LIN {X 0,Y 531.012,Z 558.342,A -85,B 0,C 180,E1 -4347.596,E2 -4347.596} C_VEL
LIN {X 0,Y 530.977,Z 558.347,A -85,B 0,C 180,E1 -4350.648,E2 -4350.648} C_VEL
LIN {X 0,Y 530.988,Z 558.345,A -85,B 0,C 180,E1 -4353.773,E2 -4353.773} C_VEL
LIN {X 0,Y 530.967,Z 558.348,A -85,B 0,C 180,E1 -4356.558,E2 -4356.558} C_VEL
LIN {X 0,Y 531.002,Z 558.343,A -85,B 0,C 180,E1 -4359.858,E2 -4359.858} C_VEL
LIN {X 0,Y 530.979,Z 558.345,A -85,B 0,C 180,E1 -4362.457,E2 -4362.457} C_VEL
LIN {X 0,Y 530.984,Z 558.347,A -85,B 0,C 180,E1 -4365.622,E2 -4365.622} C_VEL
LIN {X 0,Y 531.004,Z 558.343,A -85,B 0,C 180,E1 -4368.567,E2 -4368.567} C_VEL
LIN {X 0,Y 530.967,Z 558.349,A -85,B 0,C 180,E1 -4371.347,E2 -4371.347} C_VEL
LIN {X 0,Y 530.976,Z 558.441,A -85,B 0,C 180,E1 -4371.895,E2 -4371.895} C_VEL
LIN {X 0,Y 532.393,Z 565.517,A -85,B 0,C 180,E1 -4373.635,E2 -4373.635} C_VEL
LIN {X 0,Y 532.607,Z 569.285,A -85,B 0,C 180,E1 -4374.508,E2 -4374.508} C_VEL
LIN {X 0,Y 532.356,Z 582.925,A -85,B 0,C 180,E1 -4377.495,E2 -4377.495} C_VEL
LIN {X 0,Y 532.166,Z 596.383,A -85,B 0,C 180,E1 -4380.31,E2 -4380.31} C_VEL
LIN {X 0,Y 531.962,Z 611.243,A -85,B 0,C 180,E1 -4383.309,E2 -4383.309} C_VEL
LIN {X 0,Y 531.773,Z 627.111,A -85,B 0,C 180,E1 -4386.436,E2 -4386.436} C_VEL
LIN {X 0,Y 531.567,Z 641.948,A -85,B 0,C 180,E1 -4389.289,E2 -4389.289} C_VEL
LIN {X 0,Y 531.378,Z 654.54,A -85,B 0,C 180,E1 -4391.713,E2 -4391.713} C_VEL
LIN {X 0,Y 531.087,Z 669.174,A -85,B 0,C 180,E1 -4394.654,E2 -4394.654} C_VEL
LIN {X 0,Y 530.95,Z 678.137,A -85,B 0,C 180,E1 -4396.436,E2 -4396.436} C_VEL
LIN {X 0,Y 532.382,Z 688.546,A -85,B 0,C 180,E1 -4396.668,E2 -4396.668} C_VEL
LIN {X 0,Y 532.174,Z 700.896,A -85,B 0,C 180,E1 -4397.027,E2 -4397.027} C_VEL
LIN {X 0,Y 531.979,Z 712.521,A -85,B 0,C 180,E1 -4397.507,E2 -4397.507} C_VEL
LIN {X 0,Y 531.678,Z 724.909,A -85,B 0,C 180,E1 -4398.185,E2 -4398.185} C_VEL
LIN {X 0,Y 531.5,Z 735.754,A -85,B 0,C 180,E1 -4398.947,E2 -4398.947} C_VEL
LIN {X 0,Y 531.189,Z 746.607,A -85,B 0,C 180,E1 -4399.904,E2 -4399.904} C_VEL
LIN {X 0,Y 530.969,Z 755.419,A -85,B 0,C 180,E1 -4400.862,E2 -4400.862} C_VEL
LIN {X 0,Y 530.779,Z 764.008,A -85,B 0,C 180,E1 -4402.009,E2 -4402.009} C_VEL
LIN {X 0,Y 530.636,Z 770.872,A -85,B 0,C 180,E1 -4403.155,E2 -4403.155} C_VEL
LIN {X 0,Y 530.611,Z 776.369,A -85,B 0,C 180,E1 -4404.3,E2 -4404.3} C_VEL
LIN {X 0,Y 530.457,Z 780.679,A -85,B 0,C 180,E1 -4405.441,E2 -4405.441} C_VEL
LIN {X 0,Y 530.516,Z 782.96,A -85,B 0,C 180,E1 -4406.203,E2 -4406.203} C_VEL
LIN {X 0,Y 530.457,Z 784.809,A -85,B 0,C 180,E1 -4406.963,E2 -4406.963} C_VEL
LIN {X 0,Y 530.41,Z 786.196,A -85,B 0,C 180,E1 -4407.723,E2 -4407.723} C_VEL
LIN {X 0,Y 530.344,Z 787.786,A -85,B 0,C 180,E1 -4409.241,E2 -4409.241} C_VEL
LIN {X 0,Y 530.342,Z 788,A -85,B 0,C 180,E1 -4410.001,E2 -4410.001} C_VEL
LIN {X 0,Y 530.361,Z 787.184,A -85,B 0,C 180,E1 -4411.519,E2 -4411.519} C_VEL
LIN {X 0,Y 530.41,Z 786.196,A -85,B 0,C 180,E1 -4412.279,E2 -4412.279} C_VEL
LIN {X 0,Y 530.457,Z 784.809,A -85,B 0,C 180,E1 -4413.039,E2 -4413.039} C_VEL
LIN {X 0,Y 530.523,Z 781.893,A -85,B 0,C 180,E1 -4414.179,E2 -4414.179} C_VEL
LIN {X 0,Y 530.525,Z 777.946,A -85,B 0,C 180,E1 -4415.321,E2 -4415.321} C_VEL
LIN {X 0,Y 530.6,Z 772.262,A -85,B 0,C 180,E1 -4416.582,E2 -4416.582} C_VEL
LIN {X 0,Y 530.759,Z 765.232,A -85,B 0,C 180,E1 -4417.801,E2 -4417.801} C_VEL
LIN {X 0,Y 530.93,Z 756.987,A -85,B 0,C 180,E1 -4418.949,E2 -4418.949} C_VEL
LIN {X 0,Y 531.112,Z 748.533,A -85,B 0,C 180,E1 -4419.906,E2 -4419.906} C_VEL
LIN {X 0,Y 531.416,Z 738.086,A -85,B 0,C 180,E1 -4420.863,E2 -4420.863} C_VEL
LIN {X 0,Y 531.675,Z 727.295,A -85,B 0,C 180,E1 -4421.66,E2 -4421.66} C_VEL
LIN {X 0,Y 531.876,Z 716.394,A -85,B 0,C 180,E1 -4422.303,E2 -4422.303} C_VEL
LIN {X 0,Y 532.111,Z 704.747,A -85,B 0,C 180,E1 -4422.83,E2 -4422.83} C_VEL
LIN {X 0,Y 532.332,Z 691.322,A -85,B 0,C 180,E1 -4423.262,E2 -4423.262} C_VEL
LIN {X 0,Y 532.131,Z 685.757,A -85,B 0,C 180,E1 -4423.398,E2 -4423.398} C_VEL
LIN {X 0,Y 530.944,Z 678.031,A -85,B 0,C 180,E1 -4423.589,E2 -4423.589} C_VEL
LIN {X 0,Y 531.198,Z 663.358,A -85,B 0,C 180,E1 -4426.527,E2 -4426.527} C_VEL
LIN {X 0,Y 531.508,Z 648.458,A -85,B 0,C 180,E1 -4429.505,E2 -4429.505} C_VEL
LIN {X 0,Y 531.685,Z 632.611,A -85,B 0,C 180,E1 -4432.541,E2 -4432.541} C_VEL
LIN {X 0,Y 531.884,Z 617.998,A -85,B 0,C 180,E1 -4435.432,E2 -4435.432} C_VEL
LIN {X 0,Y 532.057,Z 605.161,A -85,B 0,C 180,E1 -4438.028,E2 -4438.028} C_VEL
LIN {X 0,Y 532.312,Z 590.837,A -85,B 0,C 180,E1 -4440.992,E2 -4440.992} C_VEL
LIN {X 0,Y 532.502,Z 577.979,A -85,B 0,C 180,E1 -4443.749,E2 -4443.749} C_VEL
LIN {X 0,Y 532.673,Z 568.114,A -85,B 0,C 180,E1 -4445.926,E2 -4445.926} C_VEL
LIN {X 0,Y 531.615,Z 561.406,A -85,B 0,C 180,E1 -4447.514,E2 -4447.514} C_VEL
LIN {X 0,Y 530.971,Z 558.349,A -85,B 0,C 180,E1 -4448.288,E2 -4448.288} C_VEL
LIN {X 0,Y 531.006,Z 558.343,A -85,B 0,C 180,E1 -4451.435,E2 -4451.435} C_VEL
LIN {X 0,Y 530.993,Z 558.346,A -85,B 0,C 180,E1 -4454.547,E2 -4454.547} C_VEL
LIN {X 0,Y 530.99,Z 558.346,A -85,B 0,C 180,E1 -4457.834,E2 -4457.834} C_VEL
LIN {X 0,Y 530.99,Z 558.344,A -85,B 0,C 180,E1 -4460.557,E2 -4460.557} C_VEL
LIN {X 0,Y 530.979,Z 558.347,A -85,B 0,C 180,E1 -4463.842,E2 -4463.842} C_VEL
LIN {X 0,Y 531.004,Z 558.342,A -85,B 0,C 180,E1 -4466.494,E2 -4466.494} C_VEL
LIN {X 0,Y 530.978,Z 558.346,A -85,B 0,C 180,E1 -4469.355,E2 -4469.355} C_VEL
LIN {X 0,Y 531.021,Z 558.34,A -85,B 0,C 180,E1 -4472.467,E2 -4472.467} C_VEL
LIN {X 0,Y 531.01,Z 558.341,A -85,B 0,C 180,E1 -4474.942,E2 -4474.942} C_VEL
LIN {X 0,Y 530.976,Z 558.346,A -85,B 0,C 180,E1 -4478.247,E2 -4478.247} C_VEL
LIN {X 0,Y 530.999,Z 558.343,A -85,B 0,C 180,E1 -4480.677,E2 -4480.677} C_VEL
LIN {X 0,Y 530.99,Z 558.343,A -85,B 0,C 180,E1 -4483.071,E2 -4483.071} C_VEL
LIN {X 0,Y 531.023,Z 558.338,A -85,B 0,C 180,E1 -4485.436,E2 -4485.436} C_VEL
LIN {X 0,Y 531.04,Z 558.339,A -85,B 0,C 180,E1 -4488.55,E2 -4488.55} C_VEL
LIN {X 0,Y 531.061,Z 558.335,A -85,B 0,C 180,E1 -4491.629,E2 -4491.629} C_VEL
LIN {X 0,Y 531.126,Z 558.327,A -85,B 0,C 180,E1 -4494.685,E2 -4494.685} C_VEL
LIN {X 0,Y 531.139,Z 558.327,A -85,B 0,C 180,E1 -4497.725,E2 -4497.725} C_VEL
LIN {X 0,Y 531.157,Z 558.324,A -85,B 0,C 180,E1 -4500.758,E2 -4500.758} C_VEL
LIN {X 0,Y 531.107,Z 558.329,A -85,B 0,C 180,E1 -4503.034,E2 -4503.034} C_VEL
LIN {X 0,Y 531.088,Z 558.333,A -85,B 0,C 180,E1 -4506.077,E2 -4506.077} C_VEL
LIN {X 0,Y 531.031,Z 558.34,A -85,B 0,C 180,E1 -4509.138,E2 -4509.138} C_VEL
LIN {X 0,Y 531.044,Z 558.337,A -85,B 0,C 180,E1 -4512.225,E2 -4512.225} C_VEL
LIN {X 0,Y 530.999,Z 558.343,A -85,B 0,C 180,E1 -4515.349,E2 -4515.349} C_VEL
LIN {X 0,Y 530.993,Z 558.345,A -85,B 0,C 180,E1 -4518.521,E2 -4518.521} C_VEL
LIN {X 0,Y 531.002,Z 558.345,A -85,B 0,C 180,E1 -4520.937,E2 -4520.937} C_VEL
LIN {X 0,Y 530.983,Z 558.345,A -85,B 0,C 180,E1 -4524.224,E2 -4524.224} C_VEL
LIN {X 0,Y 531.008,Z 558.344,A -85,B 0,C 180,E1 -4526.743,E2 -4526.743} C_VEL
LIN {X 0,Y 530.984,Z 558.345,A -85,B 0,C 180,E1 -4529.322,E2 -4529.322} C_VEL
LIN {X 0,Y 530.972,Z 558.346,A -85,B 0,C 180,E1 -4532.101,E2 -4532.101} C_VEL
LIN {X 0,Y 530.99,Z 558.346,A -85,B 0,C 180,E1 -4534.854,E2 -4534.854} C_VEL
LIN {X 0,Y 530.968,Z 558.348,A -85,B 0,C 180,E1 -4537.507,E2 -4537.507} C_VEL
LIN {X 0,Y 530.985,Z 558.345,A -85,B 0,C 180,E1 -4540.432,E2 -4540.432} C_VEL
LIN {X 0,Y 530.972,Z 558.347,A -85,B 0,C 180,E1 -4543.282,E2 -4543.282} C_VEL
LIN {X 0,Y 530.965,Z 558.347,A -85,B 0,C 180,E1 -4543.565,E2 -4543.565} C_VEL
LIN {X 0,Y 530.292,Z 558.433,A -85,B 0,C 180,E1 -4544.199,E2 -4544.199} C_VEL
LIN {X 0,Y 527.445,Z 558.788,A -85,B 0,C 180,E1 -4545.228,E2 -4545.228} C_VEL
LIN {X 0,Y 525.043,Z 559.089,A -85,B 0,C 180,E1 -4546.056,E2 -4546.056} C_VEL
LIN {X 0,Y 524.009,Z 559.216,A -85,B 0,C 180,E1 -4546.696,E2 -4546.696} C_VEL
LIN {X 0,Y 523.924,Z 559.225,A -85,B 0,C 180,E1 -4546.912,E2 -4546.912} C_VEL
LIN {X 0,Y 523.949,Z 559.22,A -85,B 0,C 180,E1 -4549.92,E2 -4549.92} C_VEL
LIN {X 0,Y 523.908,Z 559.226,A -85,B 0,C 180,E1 -4552.867,E2 -4552.867} C_VEL
LIN {X 0,Y 523.933,Z 559.222,A -85,B 0,C 180,E1 -4555.709,E2 -4555.709} C_VEL
LIN {X 0,Y 523.932,Z 559.226,A -85,B 0,C 180,E1 -4558.456,E2 -4558.456} C_VEL
LIN {X 0,Y 523.94,Z 559.221,A -85,B 0,C 180,E1 -4561.125,E2 -4561.125} C_VEL
LIN {X 0,Y 523.985,Z 559.216,A -85,B 0,C 180,E1 -4563.98,E2 -4563.98} C_VEL
LIN {X 0,Y 523.937,Z 559.223,A -85,B 0,C 180,E1 -4566.27,E2 -4566.27} C_VEL
LIN {X 0,Y 523.947,Z 559.223,A -85,B 0,C 180,E1 -4568.766,E2 -4568.766} C_VEL
LIN {X 0,Y 523.952,Z 559.222,A -85,B 0,C 180,E1 -4571.22,E2 -4571.22} C_VEL
LIN {X 0,Y 523.938,Z 559.223,A -85,B 0,C 180,E1 -4573.638,E2 -4573.638} C_VEL
LIN {X 0,Y 523.94,Z 559.224,A -85,B 0,C 180,E1 -4576.027,E2 -4576.027} C_VEL
LIN {X 0,Y 524.015,Z 559.215,A -85,B 0,C 180,E1 -4578.394,E2 -4578.394} C_VEL
LIN {X 0,Y 524.003,Z 559.215,A -85,B 0,C 180,E1 -4581.515,E2 -4581.515} C_VEL
LIN {X 0,Y 524.083,Z 559.205,A -85,B 0,C 180,E1 -4584.613,E2 -4584.613} C_VEL
LIN {X 0,Y 524.113,Z 559.203,A -85,B 0,C 180,E1 -4587.694,E2 -4587.694} C_VEL
LIN {X 0,Y 524.119,Z 559.201,A -85,B 0,C 180,E1 -4590.768,E2 -4590.768} C_VEL
LIN {X 0,Y 524.038,Z 559.227,A -85,B 0,C 180,E1 -4591.032,E2 -4591.032} C_VEL
LIN {X 0,Y 525.114,Z 563.361,A -85,B 0,C 180,E1 -4591.245,E2 -4591.245} C_VEL
LIN {X 0,Y 525.13,Z 574.326,A -85,B 0,C 180,E1 -4591.821,E2 -4591.821} C_VEL
LIN {X 0,Y 524.911,Z 584.578,A -85,B 0,C 180,E1 -4592.493,E2 -4592.493} C_VEL
LIN {X 0,Y 524.606,Z 594.134,A -85,B 0,C 180,E1 -4593.263,E2 -4593.263} C_VEL
LIN {X 0,Y 524.396,Z 603.842,A -85,B 0,C 180,E1 -4594.226,E2 -4594.226} C_VEL
LIN {X 0,Y 524.075,Z 613.228,A -85,B 0,C 180,E1 -4595.386,E2 -4595.386} C_VEL
LIN {X 0,Y 523.978,Z 619.818,A -85,B 0,C 180,E1 -4596.397,E2 -4596.397} C_VEL
LIN {X 0,Y 523.856,Z 624.671,A -85,B 0,C 180,E1 -4597.283,E2 -4597.283} C_VEL
LIN {X 0,Y 523.684,Z 630.045,A -85,B 0,C 180,E1 -4598.488,E2 -4598.488} C_VEL
LIN {X 0,Y 523.593,Z 634.07,A -85,B 0,C 180,E1 -4599.658,E2 -4599.658} C_VEL
LIN {X 0,Y 523.545,Z 637.066,A -85,B 0,C 180,E1 -4600.831,E2 -4600.831} C_VEL
LIN {X 0,Y 523.506,Z 638.563,A -85,B 0,C 180,E1 -4601.616,E2 -4601.616} C_VEL
LIN {X 0,Y 523.442,Z 640.229,A -85,B 0,C 180,E1 -4603.193,E2 -4603.193} C_VEL
LIN {X 0,Y 523.461,Z 640.494,A -85,B 0,C 180,E1 -4603.984,E2 -4603.984} C_VEL
LIN {X 0,Y 523.456,Z 639.713,A -85,B 0,C 180,E1 -4605.576,E2 -4605.576} C_VEL
LIN {X 0,Y 523.485,Z 638.737,A -85,B 0,C 180,E1 -4606.375,E2 -4606.375} C_VEL
LIN {X 0,Y 523.556,Z 636.308,A -85,B 0,C 180,E1 -4607.623,E2 -4607.623} C_VEL
LIN {X 0,Y 523.635,Z 633.025,A -85,B 0,C 180,E1 -4608.79,E2 -4608.79} C_VEL
LIN {X 0,Y 523.743,Z 628.185,A -85,B 0,C 180,E1 -4610.064,E2 -4610.064} C_VEL
LIN {X 0,Y 523.908,Z 622.475,A -85,B 0,C 180,E1 -4611.234,E2 -4611.234} C_VEL
LIN {X 0,Y 524.066,Z 616.165,A -85,B 0,C 180,E1 -4612.283,E2 -4612.283} C_VEL
LIN {X 0,Y 524.28,Z 608.781,A -85,B 0,C 180,E1 -4613.293,E2 -4613.293} C_VEL
LIN {X 0,Y 524.533,Z 600.514,A -85,B 0,C 180,E1 -4614.226,E2 -4614.226} C_VEL
LIN {X 0,Y 524.749,Z 590.363,A -85,B 0,C 180,E1 -4615.164,E2 -4615.164} C_VEL
LIN {X 0,Y 525.085,Z 578.943,A -85,B 0,C 180,E1 -4615.997,E2 -4615.997} C_VEL
LIN {X 0,Y 525.258,Z 567.57,A -85,B 0,C 180,E1 -4616.645,E2 -4616.645} C_VEL
LIN {X 0,Y 525.229,Z 563.764,A -85,B 0,C 180,E1 -4616.831,E2 -4616.831} C_VEL
LIN {X 0,Y 524.004,Z 559.217,A -85,B 0,C 180,E1 -4617.07,E2 -4617.07} C_VEL
LIN {X 0,Y 523.952,Z 559.222,A -85,B 0,C 180,E1 -4619.754,E2 -4619.754} C_VEL
LIN {X 0,Y 523.934,Z 559.223,A -85,B 0,C 180,E1 -4622.448,E2 -4622.448} C_VEL
LIN {X 0,Y 523.926,Z 559.226,A -85,B 0,C 180,E1 -4625.225,E2 -4625.225} C_VEL
LIN {X 0,Y 523.912,Z 559.226,A -85,B 0,C 180,E1 -4628.101,E2 -4628.101} C_VEL
LIN {X 0,Y 524.053,Z 559.318,A -85,B 0,C 180,E1 -4630.826,E2 -4630.826} C_VEL
LIN {X 0,Y 524.281,Z 563.958,A -85,B 0,C 180,E1 -4632.501,E2 -4632.501} C_VEL
LIN {X 0,Y 524.248,Z 571.692,A -85,B 0,C 180,E1 -4635.275,E2 -4635.275} C_VEL
LIN {X 0,Y 524.192,Z 580.087,A -85,B 0,C 180,E1 -4638.32,E2 -4638.32} C_VEL
LIN {X 0,Y 524.057,Z 587.769,A -85,B 0,C 180,E1 -4641.06,E2 -4641.06} C_VEL
LIN {X 0,Y 523.974,Z 595.445,A -85,B 0,C 180,E1 -4643.832,E2 -4643.832} C_VEL
LIN {X 0,Y 523.928,Z 602.281,A -85,B 0,C 180,E1 -4646.269,E2 -4646.269} C_VEL
LIN {X 0,Y 523.739,Z 610.522,A -85,B 0,C 180,E1 -4649.342,E2 -4649.342} C_VEL
LIN {X 0,Y 523.622,Z 618.757,A -85,B 0,C 180,E1 -4652.353,E2 -4652.353} C_VEL
LIN {X 0,Y 523.564,Z 621.51,A -85,B 0,C 180,E1 -4653.347,E2 -4653.347} C_VEL
LIN {X 0,Y 525.386,Z 632.378,A -85,B 0,C 180,E1 -4653.64,E2 -4653.64} C_VEL
LIN {X 0,Y 525.193,Z 642.791,A -85,B 0,C 180,E1 -4653.975,E2 -4653.975} C_VEL
LIN {X 0,Y 524.981,Z 652.106,A -85,B 0,C 180,E1 -4654.369,E2 -4654.369} C_VEL
LIN {X 0,Y 524.728,Z 662.67,A -85,B 0,C 180,E1 -4654.94,E2 -4654.94} C_VEL
LIN {X 0,Y 524.549,Z 671.625,A -85,B 0,C 180,E1 -4655.537,E2 -4655.537} C_VEL
LIN {X 0,Y 524.351,Z 679.01,A -85,B 0,C 180,E1 -4656.117,E2 -4656.117} C_VEL
LIN {X 0,Y 524.109,Z 687.49,A -85,B 0,C 180,E1 -4656.907,E2 -4656.907} C_VEL
LIN {X 0,Y 523.923,Z 695.109,A -85,B 0,C 180,E1 -4657.753,E2 -4657.753} C_VEL
LIN {X 0,Y 523.748,Z 701.276,A -85,B 0,C 180,E1 -4658.552,E2 -4658.552} C_VEL
LIN {X 0,Y 523.616,Z 707.87,A -85,B 0,C 180,E1 -4659.576,E2 -4659.576} C_VEL
LIN {X 0,Y 523.524,Z 712.354,A -85,B 0,C 180,E1 -4660.391,E2 -4660.391} C_VEL
LIN {X 0,Y 523.442,Z 717.73,A -85,B 0,C 180,E1 -4661.608,E2 -4661.608} C_VEL
LIN {X 0,Y 523.368,Z 721.85,A -85,B 0,C 180,E1 -4662.817,E2 -4662.817} C_VEL
LIN {X 0,Y 523.303,Z 724.035,A -85,B 0,C 180,E1 -4663.619,E2 -4663.619} C_VEL
LIN {X 0,Y 523.253,Z 725.633,A -85,B 0,C 180,E1 -4664.418,E2 -4664.418} C_VEL
LIN {X 0,Y 523.286,Z 727.629,A -85,B 0,C 180,E1 -4666.011,E2 -4666.011} C_VEL
LIN {X 0,Y 523.259,Z 727.941,A -85,B 0,C 180,E1 -4666.802,E2 -4666.802} C_VEL
LIN {X 0,Y 523.343,Z 727.386,A -85,B 0,C 180,E1 -4668.379,E2 -4668.379} C_VEL
LIN {X 0,Y 523.366,Z 726.466,A -85,B 0,C 180,E1 -4669.164,E2 -4669.164} C_VEL
LIN {X 0,Y 523.323,Z 723.382,A -85,B 0,C 180,E1 -4670.726,E2 -4670.726} C_VEL
LIN {X 0,Y 523.43,Z 719.883,A -85,B 0,C 180,E1 -4671.896,E2 -4671.896} C_VEL
LIN {X 0,Y 523.478,Z 715.303,A -85,B 0,C 180,E1 -4673.06,E2 -4673.06} C_VEL
LIN {X 0,Y 523.566,Z 710.594,A -85,B 0,C 180,E1 -4674.029,E2 -4674.029} C_VEL
LIN {X 0,Y 523.603,Z 704.939,A -85,B 0,C 180,E1 -4674.995,E2 -4674.995} C_VEL
LIN {X 0,Y 523.804,Z 698.131,A -85,B 0,C 180,E1 -4675.961,E2 -4675.961} C_VEL
LIN {X 0,Y 524.008,Z 689.945,A -85,B 0,C 180,E1 -4676.925,E2 -4676.925} C_VEL
LIN {X 0,Y 524.272,Z 681.063,A -85,B 0,C 180,E1 -4677.792,E2 -4677.792} C_VEL
LIN {X 0,Y 524.46,Z 672.831,A -85,B 0,C 180,E1 -4678.465,E2 -4678.465} C_VEL
LIN {X 0,Y 524.686,Z 664.45,A -85,B 0,C 180,E1 -4679.041,E2 -4679.041} C_VEL
LIN {X 0,Y 524.901,Z 656.14,A -85,B 0,C 180,E1 -4679.521,E2 -4679.521} C_VEL
LIN {X 0,Y 525.152,Z 645.757,A -85,B 0,C 180,E1 -4680,E2 -4680} C_VEL
LIN {X 0,Y 525.326,Z 634.77,A -85,B 0,C 180,E1 -4680.384,E2 -4680.384} C_VEL
LIN {X 0,Y 525.026,Z 630.01,A -85,B 0,C 180,E1 -4680.528,E2 -4680.528} C_VEL
LIN {X 0,Y 523.568,Z 621.481,A -85,B 0,C 180,E1 -4680.769,E2 -4680.769} C_VEL
LIN {X 0,Y 523.743,Z 614.266,A -85,B 0,C 180,E1 -4683.462,E2 -4683.462} C_VEL
LIN {X 0,Y 523.808,Z 607.857,A -85,B 0,C 180,E1 -4685.776,E2 -4685.776} C_VEL
LIN {X 0,Y 523.962,Z 600.52,A -85,B 0,C 180,E1 -4688.485,E2 -4688.485} C_VEL
LIN {X 0,Y 524.052,Z 591.747,A -85,B 0,C 180,E1 -4691.605,E2 -4691.605} C_VEL
LIN {X 0,Y 524.082,Z 583.632,A -85,B 0,C 180,E1 -4694.365,E2 -4694.365} C_VEL
LIN {X 0,Y 524.078,Z 575.146,A -85,B 0,C 180,E1 -4697.159,E2 -4697.159} C_VEL
LIN {X 0,Y 523.94,Z 565.718,A -85,B 0,C 180,E1 -4700.125,E2 -4700.125} C_VEL
LIN {X 0,Y 523.928,Z 559.227,A -85,B 0,C 180,E1 -4702.061,E2 -4702.061} C_VEL
LIN {X 0,Y 523.931,Z 559.226,A -85,B 0,C 180,E1 -4704.572,E2 -4704.572} C_VEL
LIN {X 0,Y 523.952,Z 559.223,A -85,B 0,C 180,E1 -4707.133,E2 -4707.133} C_VEL
LIN {X 0,Y 523.951,Z 559.222,A -85,B 0,C 180,E1 -4709.756,E2 -4709.756} C_VEL
LIN {X 0,Y 523.935,Z 559.224,A -85,B 0,C 180,E1 -4712.45,E2 -4712.45} C_VEL
LIN {X 0,Y 523.932,Z 559.225,A -85,B 0,C 180,E1 -4715.226,E2 -4715.226} C_VEL
LIN {X 0,Y 523.915,Z 559.226,A -85,B 0,C 180,E1 -4718.102,E2 -4718.102} C_VEL
LIN {X 0,Y 523.957,Z 559.221,A -85,B 0,C 180,E1 -4721.091,E2 -4721.091} C_VEL
LIN {X 0,Y 523.937,Z 559.222,A -85,B 0,C 180,E1 -4724.229,E2 -4724.229} C_VEL
LIN {X 0,Y 523.922,Z 559.226,A -85,B 0,C 180,E1 -4726.835,E2 -4726.835} C_VEL
LIN {X 0,Y 523.976,Z 559.22,A -85,B 0,C 180,E1 -4729.924,E2 -4729.924} C_VEL
LIN {X 0,Y 523.944,Z 559.413,A -85,B 0,C 180,E1 -4731.657,E2 -4731.657} C_VEL
LIN {X 0,Y 525.547,Z 567.486,A -85,B 0,C 180,E1 -4733.678,E2 -4733.678} C_VEL
LIN {X 0,Y 525.601,Z 573.801,A -85,B 0,C 180,E1 -4735.138,E2 -4735.138} C_VEL
LIN {X 0,Y 525.359,Z 586.217,A -85,B 0,C 180,E1 -4737.877,E2 -4737.877} C_VEL
LIN {X 0,Y 525.163,Z 598.325,A -85,B 0,C 180,E1 -4740.443,E2 -4740.443} C_VEL
LIN {X 0,Y 524.916,Z 612.503,A -85,B 0,C 180,E1 -4743.352,E2 -4743.352} C_VEL
LIN {X 0,Y 524.713,Z 627.296,A -85,B 0,C 180,E1 -4746.309,E2 -4746.309} C_VEL
LIN {X 0,Y 524.501,Z 642.061,A -85,B 0,C 180,E1 -4749.202,E2 -4749.202} C_VEL
LIN {X 0,Y 524.272,Z 657.347,A -85,B 0,C 180,E1 -4752.134,E2 -4752.134} C_VEL
LIN {X 0,Y 524.039,Z 670.868,A -85,B 0,C 180,E1 -4754.786,E2 -4754.786} C_VEL
LIN {X 0,Y 523.899,Z 678.137,A -85,B 0,C 180,E1 -4756.25,E2 -4756.25} C_VEL
LIN {X 0,Y 525.463,Z 688.545,A -85,B 0,C 180,E1 -4756.489,E2 -4756.489} C_VEL
LIN {X 0,Y 525.247,Z 700.895,A -85,B 0,C 180,E1 -4756.853,E2 -4756.853} C_VEL
LIN {X 0,Y 525.054,Z 712.52,A -85,B 0,C 180,E1 -4757.34,E2 -4757.34} C_VEL
LIN {X 0,Y 524.718,Z 723.969,A -85,B 0,C 180,E1 -4757.967,E2 -4757.967} C_VEL
LIN {X 0,Y 524.547,Z 734.496,A -85,B 0,C 180,E1 -4758.701,E2 -4758.701} C_VEL
LIN {X 0,Y 524.227,Z 744.654,A -85,B 0,C 180,E1 -4759.574,E2 -4759.574} C_VEL
LIN {X 0,Y 523.971,Z 753.792,A -85,B 0,C 180,E1 -4760.544,E2 -4760.544} C_VEL
LIN {X 0,Y 523.759,Z 762.693,A -85,B 0,C 180,E1 -4761.707,E2 -4761.707} C_VEL
LIN {X 0,Y 523.583,Z 769.853,A -85,B 0,C 180,E1 -4762.868,E2 -4762.868} C_VEL
LIN {X 0,Y 523.544,Z 776.369,A -85,B 0,C 180,E1 -4764.222,E2 -4764.222} C_VEL
LIN {X 0,Y 523.361,Z 780.679,A -85,B 0,C 180,E1 -4765.379,E2 -4765.379} C_VEL
LIN {X 0,Y 523.443,Z 782.96,A -85,B 0,C 180,E1 -4766.151,E2 -4766.151} C_VEL
LIN {X 0,Y 523.367,Z 784.809,A -85,B 0,C 180,E1 -4766.922,E2 -4766.922} C_VEL
LIN {X 0,Y 523.334,Z 786.195,A -85,B 0,C 180,E1 -4767.692,E2 -4767.692} C_VEL
LIN {X 0,Y 523.25,Z 787.786,A -85,B 0,C 180,E1 -4769.231,E2 -4769.231} C_VEL
LIN {X 0,Y 523.246,Z 788,A -85,B 0,C 180,E1 -4770.001,E2 -4770.001} C_VEL
LIN {X 0,Y 523.274,Z 787.183,A -85,B 0,C 180,E1 -4771.54,E2 -4771.54} C_VEL
LIN {X 0,Y 523.334,Z 786.196,A -85,B 0,C 180,E1 -4772.31,E2 -4772.31} C_VEL
LIN {X 0,Y 523.368,Z 784.809,A -85,B 0,C 180,E1 -4773.08,E2 -4773.08} C_VEL
LIN {X 0,Y 523.442,Z 781.893,A -85,B 0,C 180,E1 -4774.236,E2 -4774.236} C_VEL
LIN {X 0,Y 523.464,Z 777.946,A -85,B 0,C 180,E1 -4775.393,E2 -4775.393} C_VEL
LIN {X 0,Y 523.524,Z 772.726,A -85,B 0,C 180,E1 -4776.581,E2 -4776.581} C_VEL
LIN {X 0,Y 523.666,Z 766.463,A -85,B 0,C 180,E1 -4777.713,E2 -4777.713} C_VEL
LIN {X 0,Y 523.856,Z 758.472,A -85,B 0,C 180,E1 -4778.876,E2 -4778.876} C_VEL
LIN {X 0,Y 524.085,Z 750.327,A -85,B 0,C 180,E1 -4779.845,E2 -4779.845} C_VEL
LIN {X 0,Y 524.356,Z 740.391,A -85,B 0,C 180,E1 -4780.816,E2 -4780.816} C_VEL
LIN {X 0,Y 524.708,Z 729.123,A -85,B 0,C 180,E1 -4781.692,E2 -4781.692} C_VEL
LIN {X 0,Y 524.902,Z 718.16,A -85,B 0,C 180,E1 -4782.371,E2 -4782.371} C_VEL
LIN {X 0,Y 525.179,Z 705.958,A -85,B 0,C 180,E1 -4782.954,E2 -4782.954} C_VEL
LIN {X 0,Y 525.383,Z 693.15,A -85,B 0,C 180,E1 -4783.391,E2 -4783.391} C_VEL
LIN {X 0,Y 525.25,Z 686.637,A -85,B 0,C 180,E1 -4783.558,E2 -4783.558} C_VEL
LIN {X 0,Y 523.895,Z 678.031,A -85,B 0,C 180,E1 -4783.776,E2 -4783.776} C_VEL
LIN {X 0,Y 524.176,Z 663.237,A -85,B 0,C 180,E1 -4786.755,E2 -4786.755} C_VEL
LIN {X 0,Y 524.425,Z 648.622,A -85,B 0,C 180,E1 -4789.575,E2 -4789.575} C_VEL
LIN {X 0,Y 524.618,Z 633.045,A -85,B 0,C 180,E1 -4792.6,E2 -4792.6} C_VEL
LIN {X 0,Y 524.879,Z 618.272,A -85,B 0,C 180,E1 -4795.584,E2 -4795.584} C_VEL
LIN {X 0,Y 525.128,Z 603.666,A -85,B 0,C 180,E1 -4798.585,E2 -4798.585} C_VEL
LIN {X 0,Y 525.395,Z 589.108,A -85,B 0,C 180,E1 -4801.671,E2 -4801.671} C_VEL
LIN {X 0,Y 525.62,Z 575.612,A -85,B 0,C 180,E1 -4804.63,E2 -4804.63} C_VEL
LIN {X 0,Y 525.609,Z 568.079,A -85,B 0,C 180,E1 -4806.328,E2 -4806.328} C_VEL
LIN {X 0,Y 523.922,Z 559.227,A -85,B 0,C 180,E1 -4808.53,E2 -4808.53} C_VEL
LIN {X 0,Y 523.967,Z 559.22,A -85,B 0,C 180,E1 -4811.311,E2 -4811.311} C_VEL
LIN {X 0,Y 523.961,Z 559.221,A -85,B 0,C 180,E1 -4814.691,E2 -4814.691} C_VEL
LIN {X 0,Y 523.959,Z 559.222,A -85,B 0,C 180,E1 -4817.881,E2 -4817.881} C_VEL
LIN {X 0,Y 523.924,Z 559.224,A -85,B 0,C 180,E1 -4820.915,E2 -4820.915} C_VEL
LIN {X 0,Y 523.933,Z 559.225,A -85,B 0,C 180,E1 -4823.828,E2 -4823.828} C_VEL
LIN {X 0,Y 523.946,Z 559.221,A -85,B 0,C 180,E1 -4826.636,E2 -4826.636} C_VEL
LIN {X 0,Y 523.96,Z 559.22,A -85,B 0,C 180,E1 -4829.356,E2 -4829.356} C_VEL
LIN {X 0,Y 523.984,Z 559.217,A -85,B 0,C 180,E1 -4832.281,E2 -4832.281} C_VEL
LIN {X 0,Y 523.957,Z 559.22,A -85,B 0,C 180,E1 -4834.581,E2 -4834.581} C_VEL
LIN {X 0,Y 523.916,Z 559.224,A -85,B 0,C 180,E1 -4837.106,E2 -4837.106} C_VEL
LIN {X 0,Y 523.983,Z 559.217,A -85,B 0,C 180,E1 -4839.866,E2 -4839.866} C_VEL
LIN {X 0,Y 523.971,Z 559.218,A -85,B 0,C 180,E1 -4842.837,E2 -4842.837} C_VEL
LIN {X 0,Y 523.981,Z 559.216,A -85,B 0,C 180,E1 -4845.236,E2 -4845.236} C_VEL
LIN {X 0,Y 524.017,Z 559.215,A -85,B 0,C 180,E1 -4848.394,E2 -4848.394} C_VEL
LIN {X 0,Y 524.009,Z 559.213,A -85,B 0,C 180,E1 -4851.516,E2 -4851.516} C_VEL
LIN {X 0,Y 524.087,Z 559.204,A -85,B 0,C 180,E1 -4854.613,E2 -4854.613} C_VEL
LIN {X 0,Y 524.112,Z 559.202,A -85,B 0,C 180,E1 -4857.694,E2 -4857.694} C_VEL
LIN {X 0,Y 524.128,Z 559.199,A -85,B 0,C 180,E1 -4860.768,E2 -4860.768} C_VEL
LIN {X 0,Y 524.074,Z 559.205,A -85,B 0,C 180,E1 -4863.075,E2 -4863.075} C_VEL
LIN {X 0,Y 524.05,Z 559.209,A -85,B 0,C 180,E1 -4866.159,E2 -4866.159} C_VEL
LIN {X 0,Y 523.999,Z 559.216,A -85,B 0,C 180,E1 -4869.262,E2 -4869.262} C_VEL
LIN {X 0,Y 524.006,Z 559.215,A -85,B 0,C 180,E1 -4871.739,E2 -4871.739} C_VEL
LIN {X 0,Y 523.996,Z 559.217,A -85,B 0,C 180,E1 -4875.052,E2 -4875.052} C_VEL
LIN {X 0,Y 523.967,Z 559.219,A -85,B 0,C 180,E1 -4877.969,E2 -4877.969} C_VEL
LIN {X 0,Y 523.975,Z 559.218,A -85,B 0,C 180,E1 -4880.41,E2 -4880.41} C_VEL
LIN {X 0,Y 523.919,Z 559.225,A -85,B 0,C 180,E1 -4882.893,E2 -4882.893} C_VEL
LIN {X 0,Y 523.955,Z 559.22,A -85,B 0,C 180,E1 -4885.418,E2 -4885.418} C_VEL
LIN {X 0,Y 523.972,Z 559.219,A -85,B 0,C 180,E1 -4887.998,E2 -4887.998} C_VEL
LIN {X 0,Y 523.946,Z 559.221,A -85,B 0,C 180,E1 -4890.854,E2 -4890.854} C_VEL
LIN {X 0,Y 523.963,Z 559.219,A -85,B 0,C 180,E1 -4893.734,E2 -4893.734} C_VEL
LIN {X 0,Y 523.925,Z 559.226,A -85,B 0,C 180,E1 -4896.404,E2 -4896.404} C_VEL
LIN {X 0,Y 523.924,Z 559.224,A -85,B 0,C 180,E1 -4899.084,E2 -4899.084} C_VEL
LIN {X 0,Y 523.958,Z 559.222,A -85,B 0,C 180,E1 -4902.118,E2 -4902.118} C_VEL
LIN {X 0,Y 523.958,Z 559.221,A -85,B 0,C 180,E1 -4905.308,E2 -4905.308} C_VEL
LIN {X 0,Y 523.924,Z 559.225,A -85,B 0,C 180,E1 -4906.912,E2 -4906.912} C_VEL
LIN {X 0,Y 523.257,Z 559.307,A -85,B 0,C 180,E1 -4907.554,E2 -4907.554} C_VEL
LIN {X 0,Y 520.412,Z 559.664,A -85,B 0,C 180,E1 -4908.595,E2 -4908.595} C_VEL
LIN {X 0,Y 518.006,Z 559.967,A -85,B 0,C 180,E1 -4909.434,E2 -4909.434} C_VEL
LIN {X 0,Y 516.969,Z 560.094,A -85,B 0,C 180,E1 -4910.082,E2 -4910.082} C_VEL
LIN {X 0,Y 516.883,Z 560.104,A -85,B 0,C 180,E1 -4910.301,E2 -4910.301} C_VEL
LIN {X 0,Y 516.877,Z 560.102,A -85,B 0,C 180,E1 -4913.343,E2 -4913.343} C_VEL
LIN {X 0,Y 516.908,Z 560.1,A -85,B 0,C 180,E1 -4916.12,E2 -4916.12} C_VEL
LIN {X 0,Y 516.893,Z 560.1,A -85,B 0,C 180,E1 -4918.935,E2 -4918.935} C_VEL
LIN {X 0,Y 516.92,Z 560.096,A -85,B 0,C 180,E1 -4921.584,E2 -4921.584} C_VEL
LIN {X 0,Y 516.932,Z 560.097,A -85,B 0,C 180,E1 -4924.21,E2 -4924.21} C_VEL
LIN {X 0,Y 516.873,Z 560.103,A -85,B 0,C 180,E1 -4926.776,E2 -4926.776} C_VEL
LIN {X 0,Y 516.94,Z 560.093,A -85,B 0,C 180,E1 -4929.731,E2 -4929.731} C_VEL
LIN {X 0,Y 516.93,Z 560.097,A -85,B 0,C 180,E1 -4932.596,E2 -4932.596} C_VEL
LIN {X 0,Y 516.942,Z 560.094,A -85,B 0,C 180,E1 -4935.03,E2 -4935.03} C_VEL
LIN {X 0,Y 517.004,Z 560.088,A -85,B 0,C 180,E1 -4938.234,E2 -4938.234} C_VEL
LIN {X 0,Y 516.968,Z 560.091,A -85,B 0,C 180,E1 -4941.399,E2 -4941.399} C_VEL
LIN {X 0,Y 517.01,Z 560.084,A -85,B 0,C 180,E1 -4943.756,E2 -4943.756} C_VEL
LIN {X 0,Y 517.085,Z 560.079,A -85,B 0,C 180,E1 -4947.662,E2 -4947.662} C_VEL
LIN {X 0,Y 517.09,Z 560.077,A -85,B 0,C 180,E1 -4950.778,E2 -4950.778} C_VEL
LIN {X 0,Y 517.077,Z 560.168,A -85,B 0,C 180,E1 -4950.851,E2 -4950.851} C_VEL
LIN {X 0,Y 518.448,Z 566.112,A -85,B 0,C 180,E1 -4951.164,E2 -4951.164} C_VEL
LIN {X 0,Y 518.253,Z 576.837,A -85,B 0,C 180,E1 -4951.748,E2 -4951.748} C_VEL
LIN {X 0,Y 517.926,Z 588.106,A -85,B 0,C 180,E1 -4952.527,E2 -4952.527} C_VEL
LIN {X 0,Y 517.613,Z 599.227,A -85,B 0,C 180,E1 -4953.502,E2 -4953.502} C_VEL
LIN {X 0,Y 517.362,Z 608.127,A -85,B 0,C 180,E1 -4954.479,E2 -4954.479} C_VEL
LIN {X 0,Y 517.127,Z 615.497,A -85,B 0,C 180,E1 -4955.458,E2 -4955.458} C_VEL
LIN {X 0,Y 517.006,Z 621.924,A -85,B 0,C 180,E1 -4956.493,E2 -4956.493} C_VEL
LIN {X 0,Y 516.85,Z 626.758,A -85,B 0,C 180,E1 -4957.421,E2 -4957.421} C_VEL
LIN {X 0,Y 516.686,Z 631.739,A -85,B 0,C 180,E1 -4958.604,E2 -4958.604} C_VEL
LIN {X 0,Y 516.579,Z 635.606,A -85,B 0,C 180,E1 -4959.791,E2 -4959.791} C_VEL
LIN {X 0,Y 516.513,Z 638.453,A -85,B 0,C 180,E1 -4960.981,E2 -4960.981} C_VEL
LIN {X 0,Y 516.47,Z 639.849,A -85,B 0,C 180,E1 -4961.777,E2 -4961.777} C_VEL
LIN {X 0,Y 516.43,Z 640.792,A -85,B 0,C 180,E1 -4962.576,E2 -4962.576} C_VEL
LIN {X 0,Y 516.431,Z 641.491,A -85,B 0,C 180,E1 -4964.178,E2 -4964.178} C_VEL
LIN {X 0,Y 516.438,Z 641.215,A -85,B 0,C 180,E1 -4964.984,E2 -4964.984} C_VEL
LIN {X 0,Y 516.476,Z 639.437,A -85,B 0,C 180,E1 -4966.603,E2 -4966.603} C_VEL
LIN {X 0,Y 516.546,Z 637.137,A -85,B 0,C 180,E1 -4967.75,E2 -4967.75} C_VEL
LIN {X 0,Y 516.662,Z 633.359,A -85,B 0,C 180,E1 -4969.053,E2 -4969.053} C_VEL
LIN {X 0,Y 516.784,Z 628.205,A -85,B 0,C 180,E1 -4970.371,E2 -4970.371} C_VEL
LIN {X 0,Y 516.982,Z 622.398,A -85,B 0,C 180,E1 -4971.533,E2 -4971.533} C_VEL
LIN {X 0,Y 517.134,Z 616.756,A -85,B 0,C 180,E1 -4972.462,E2 -4972.462} C_VEL
LIN {X 0,Y 517.352,Z 609.87,A -85,B 0,C 180,E1 -4973.412,E2 -4973.412} C_VEL
LIN {X 0,Y 517.645,Z 600.936,A -85,B 0,C 180,E1 -4974.427,E2 -4974.427} C_VEL
LIN {X 0,Y 517.86,Z 591.462,A -85,B 0,C 180,E1 -4975.308,E2 -4975.308} C_VEL
LIN {X 0,Y 518.218,Z 580.39,A -85,B 0,C 180,E1 -4976.131,E2 -4976.131} C_VEL
LIN {X 0,Y 518.41,Z 567.979,A -85,B 0,C 180,E1 -4976.846,E2 -4976.846} C_VEL
LIN {X 0,Y 518.152,Z 564.511,A -85,B 0,C 180,E1 -4977.024,E2 -4977.024} C_VEL
LIN {X 0,Y 516.949,Z 560.095,A -85,B 0,C 180,E1 -4977.27,E2 -4977.27} C_VEL
LIN {X 0,Y 516.897,Z 560.101,A -85,B 0,C 180,E1 -4980.202,E2 -4980.202} C_VEL
LIN {X 0,Y 516.892,Z 560.102,A -85,B 0,C 180,E1 -4982.946,E2 -4982.946} C_VEL
LIN {X 0,Y 516.882,Z 560.101,A -85,B 0,C 180,E1 -4985.778,E2 -4985.778} C_VEL
LIN {X 0,Y 516.913,Z 560.098,A -85,B 0,C 180,E1 -4989.198,E2 -4989.198} C_VEL
LIN {X 0,Y 517.02,Z 560.263,A -85,B 0,C 180,E1 -4990.727,E2 -4990.727} C_VEL
LIN {X 0,Y 517.3,Z 564.45,A -85,B 0,C 180,E1 -4992.259,E2 -4992.259} C_VEL
LIN {X 0,Y 517.242,Z 572.183,A -85,B 0,C 180,E1 -4995.046,E2 -4995.046} C_VEL
LIN {X 0,Y 517.204,Z 579.568,A -85,B 0,C 180,E1 -4997.73,E2 -4997.73} C_VEL
LIN {X 0,Y 517.088,Z 586.67,A -85,B 0,C 180,E1 -5000.298,E2 -5000.298} C_VEL
LIN {X 0,Y 516.963,Z 594.988,A -85,B 0,C 180,E1 -5003.328,E2 -5003.328} C_VEL
LIN {X 0,Y 516.889,Z 602.693,A -85,B 0,C 180,E1 -5006.12,E2 -5006.12} C_VEL
LIN {X 0,Y 516.703,Z 610.365,A -85,B 0,C 180,E1 -5008.968,E2 -5008.968} C_VEL
LIN {X 0,Y 516.584,Z 617.348,A -85,B 0,C 180,E1 -5011.565,E2 -5011.565} C_VEL
LIN {X 0,Y 516.506,Z 621.677,A -85,B 0,C 180,E1 -5013.154,E2 -5013.154} C_VEL
LIN {X 0,Y 518.431,Z 632.976,A -85,B 0,C 180,E1 -5013.469,E2 -5013.469} C_VEL
LIN {X 0,Y 518.283,Z 643.121,A -85,B 0,C 180,E1 -5013.805,E2 -5013.805} C_VEL
LIN {X 0,Y 518.072,Z 652.032,A -85,B 0,C 180,E1 -5014.187,E2 -5014.187} C_VEL
LIN {X 0,Y 517.85,Z 661.417,A -85,B 0,C 180,E1 -5014.691,E2 -5014.691} C_VEL
LIN {X 0,Y 517.577,Z 671.564,A -85,B 0,C 180,E1 -5015.37,E2 -5015.37} C_VEL
LIN {X 0,Y 517.317,Z 680.026,A -85,B 0,C 180,E1 -5016.055,E2 -5016.055} C_VEL
LIN {X 0,Y 517.1,Z 687.667,A -85,B 0,C 180,E1 -5016.788,E2 -5016.788} C_VEL
LIN {X 0,Y 516.904,Z 695.085,A -85,B 0,C 180,E1 -5017.623,E2 -5017.623} C_VEL
LIN {X 0,Y 516.69,Z 701.391,A -85,B 0,C 180,E1 -5018.454,E2 -5018.454} C_VEL
LIN {X 0,Y 516.579,Z 706.817,A -85,B 0,C 180,E1 -5019.285,E2 -5019.285} C_VEL
LIN {X 0,Y 516.435,Z 713.377,A -85,B 0,C 180,E1 -5020.524,E2 -5020.524} C_VEL
LIN {X 0,Y 516.381,Z 717.045,A -85,B 0,C 180,E1 -5021.347,E2 -5021.347} C_VEL
LIN {X 0,Y 516.287,Z 721.334,A -85,B 0,C 180,E1 -5022.574,E2 -5022.574} C_VEL
LIN {X 0,Y 516.243,Z 723.584,A -85,B 0,C 180,E1 -5023.388,E2 -5023.388} C_VEL
LIN {X 0,Y 516.199,Z 726.589,A -85,B 0,C 180,E1 -5025.008,E2 -5025.008} C_VEL
LIN {X 0,Y 516.182,Z 727.507,A -85,B 0,C 180,E1 -5025.814,E2 -5025.814} C_VEL
LIN {X 0,Y 516.17,Z 727.886,A -85,B 0,C 180,E1 -5027.418,E2 -5027.418} C_VEL
LIN {X 0,Y 516.27,Z 727.198,A -85,B 0,C 180,E1 -5028.555,E2 -5028.555} C_VEL
LIN {X 0,Y 516.258,Z 725.435,A -85,B 0,C 180,E1 -5029.807,E2 -5029.807} C_VEL
LIN {X 0,Y 516.277,Z 722.776,A -85,B 0,C 180,E1 -5030.994,E2 -5030.994} C_VEL
LIN {X 0,Y 516.354,Z 719.098,A -85,B 0,C 180,E1 -5032.178,E2 -5032.178} C_VEL
LIN {X 0,Y 516.431,Z 714.019,A -85,B 0,C 180,E1 -5033.424,E2 -5033.424} C_VEL
LIN {X 0,Y 516.514,Z 709.402,A -85,B 0,C 180,E1 -5034.339,E2 -5034.339} C_VEL
LIN {X 0,Y 516.577,Z 704.808,A -85,B 0,C 180,E1 -5035.123,E2 -5035.123} C_VEL
LIN {X 0,Y 516.756,Z 697.985,A -85,B 0,C 180,E1 -5036.101,E2 -5036.101} C_VEL
LIN {X 0,Y 516.932,Z 691.603,A -85,B 0,C 180,E1 -5036.883,E2 -5036.883} C_VEL
LIN {X 0,Y 517.224,Z 683.068,A -85,B 0,C 180,E1 -5037.761,E2 -5037.761} C_VEL
LIN {X 0,Y 517.468,Z 673.973,A -85,B 0,C 180,E1 -5038.541,E2 -5038.541} C_VEL
LIN {X 0,Y 517.757,Z 664.286,A -85,B 0,C 180,E1 -5039.223,E2 -5039.223} C_VEL
LIN {X 0,Y 518.047,Z 653.99,A -85,B 0,C 180,E1 -5039.806,E2 -5039.806} C_VEL
LIN {X 0,Y 518.33,Z 644.187,A -85,B 0,C 180,E1 -5040.243,E2 -5040.243} C_VEL
LIN {X 0,Y 518.442,Z 633.487,A -85,B 0,C 180,E1 -5040.607,E2 -5040.607} C_VEL
LIN {X 0,Y 516.855,Z 623.448,A -85,B 0,C 180,E1 -5040.892,E2 -5040.892} C_VEL
LIN {X 0,Y 516.554,Z 621.883,A -85,B 0,C 180,E1 -5040.95,E2 -5040.95} C_VEL
LIN {X 0,Y 516.671,Z 614.054,A -85,B 0,C 180,E1 -5043.9,E2 -5043.9} C_VEL
LIN {X 0,Y 516.771,Z 608.623,A -85,B 0,C 180,E1 -5045.855,E2 -5045.855} C_VEL
LIN {X 0,Y 516.935,Z 601.101,A -85,B 0,C 180,E1 -5048.601,E2 -5048.601} C_VEL
LIN {X 0,Y 516.985,Z 593.293,A -85,B 0,C 180,E1 -5051.369,E2 -5051.369} C_VEL
LIN {X 0,Y 517.041,Z 587.591,A -85,B 0,C 180,E1 -5053.361,E2 -5053.361} C_VEL
LIN {X 0,Y 517.046,Z 579.174,A -85,B 0,C 180,E1 -5056.18,E2 -5056.18} C_VEL
LIN {X 0,Y 516.992,Z 571.589,A -85,B 0,C 180,E1 -5058.631,E2 -5058.631} C_VEL
LIN {X 0,Y 516.919,Z 562.142,A -85,B 0,C 180,E1 -5061.537,E2 -5061.537} C_VEL
LIN {X 0,Y 516.884,Z 560.104,A -85,B 0,C 180,E1 -5062.168,E2 -5062.168} C_VEL
LIN {X 0,Y 516.906,Z 560.103,A -85,B 0,C 180,E1 -5064.929,E2 -5064.929} C_VEL
LIN {X 0,Y 516.922,Z 560.099,A -85,B 0,C 180,E1 -5067.907,E2 -5067.907} C_VEL
LIN {X 0,Y 516.897,Z 560.102,A -85,B 0,C 180,E1 -5070.204,E2 -5070.204} C_VEL
LIN {X 0,Y 516.893,Z 560.101,A -85,B 0,C 180,E1 -5072.947,E2 -5072.947} C_VEL
LIN {X 0,Y 516.888,Z 560.101,A -85,B 0,C 180,E1 -5075.779,E2 -5075.779} C_VEL
LIN {X 0,Y 516.883,Z 560.102,A -85,B 0,C 180,E1 -5078.716,E2 -5078.716} C_VEL
LIN {X 0,Y 516.915,Z 560.096,A -85,B 0,C 180,E1 -5081.775,E2 -5081.775} C_VEL
LIN {X 0,Y 516.919,Z 560.098,A -85,B 0,C 180,E1 -5085.011,E2 -5085.011} C_VEL
LIN {X 0,Y 516.92,Z 560.096,A -85,B 0,C 180,E1 -5088.398,E2 -5088.398} C_VEL
LIN {X 0,Y 516.918,Z 560.3,A -85,B 0,C 180,E1 -5091.385,E2 -5091.385} C_VEL
LIN {X 0,Y 518.674,Z 569.122,A -85,B 0,C 180,E1 -5093.645,E2 -5093.645} C_VEL
LIN {X 0,Y 518.661,Z 576.274,A -85,B 0,C 180,E1 -5095.313,E2 -5095.313} C_VEL
LIN {X 0,Y 518.358,Z 588.643,A -85,B 0,C 180,E1 -5098.079,E2 -5098.079} C_VEL
LIN {X 0,Y 518.093,Z 602.204,A -85,B 0,C 180,E1 -5100.992,E2 -5100.992} C_VEL
LIN {X 0,Y 517.884,Z 616.347,A -85,B 0,C 180,E1 -5103.926,E2 -5103.926} C_VEL
LIN {X 0,Y 517.603,Z 632.384,A -85,B 0,C 180,E1 -5107.162,E2 -5107.162} C_VEL
LIN {X 0,Y 517.352,Z 648.547,A -85,B 0,C 180,E1 -5110.354,E2 -5110.354} C_VEL
LIN {X 0,Y 517.103,Z 663.283,A -85,B 0,C 180,E1 -5113.214,E2 -5113.214} C_VEL
LIN {X 0,Y 516.85,Z 677.981,A -85,B 0,C 180,E1 -5116.059,E2 -5116.059} C_VEL
LIN {X 0,Y 518.578,Z 689.542,A -85,B 0,C 180,E1 -5116.331,E2 -5116.331} C_VEL
LIN {X 0,Y 518.319,Z 702.195,A -85,B 0,C 180,E1 -5116.724,E2 -5116.724} C_VEL
LIN {X 0,Y 518.055,Z 714.505,A -85,B 0,C 180,E1 -5117.265,E2 -5117.265} C_VEL
LIN {X 0,Y 517.723,Z 726.593,A -85,B 0,C 180,E1 -5117.972,E2 -5117.972} C_VEL
LIN {X 0,Y 517.473,Z 738.101,A -85,B 0,C 180,E1 -5118.842,E2 -5118.842} C_VEL
LIN {X 0,Y 517.079,Z 748.547,A -85,B 0,C 180,E1 -5119.824,E2 -5119.824} C_VEL
LIN {X 0,Y 516.867,Z 756.998,A -85,B 0,C 180,E1 -5120.807,E2 -5120.807} C_VEL
LIN {X 0,Y 516.64,Z 765.24,A -85,B 0,C 180,E1 -5121.986,E2 -5121.986} C_VEL
LIN {X 0,Y 516.479,Z 772.081,A -85,B 0,C 180,E1 -5123.202,E2 -5123.202} C_VEL
LIN {X 0,Y 516.405,Z 777.952,A -85,B 0,C 180,E1 -5124.534,E2 -5124.534} C_VEL
LIN {X 0,Y 516.343,Z 781.896,A -85,B 0,C 180,E1 -5125.708,E2 -5125.708} C_VEL
LIN {X 0,Y 516.282,Z 784.808,A -85,B 0,C 180,E1 -5126.879,E2 -5126.879} C_VEL
LIN {X 0,Y 516.26,Z 786.194,A -85,B 0,C 180,E1 -5127.66,E2 -5127.66} C_VEL
LIN {X 0,Y 516.16,Z 787.786,A -85,B 0,C 180,E1 -5129.221,E2 -5129.221} C_VEL
LIN {X 0,Y 516.154,Z 788,A -85,B 0,C 180,E1 -5130.001,E2 -5130.001} C_VEL
LIN {X 0,Y 516.192,Z 787.183,A -85,B 0,C 180,E1 -5131.561,E2 -5131.561} C_VEL
LIN {X 0,Y 516.26,Z 786.195,A -85,B 0,C 180,E1 -5132.341,E2 -5132.341} C_VEL
LIN {X 0,Y 516.283,Z 784.809,A -85,B 0,C 180,E1 -5133.122,E2 -5133.122} C_VEL
LIN {X 0,Y 516.344,Z 781.893,A -85,B 0,C 180,E1 -5134.294,E2 -5134.294} C_VEL
LIN {X 0,Y 516.406,Z 777.946,A -85,B 0,C 180,E1 -5135.467,E2 -5135.467} C_VEL
LIN {X 0,Y 516.487,Z 772.031,A -85,B 0,C 180,E1 -5136.808,E2 -5136.808} C_VEL
LIN {X 0,Y 516.642,Z 765.231,A -85,B 0,C 180,E1 -5138.016,E2 -5138.016} C_VEL
LIN {X 0,Y 516.87,Z 756.987,A -85,B 0,C 180,E1 -5139.194,E2 -5139.194} C_VEL
LIN {X 0,Y 517.079,Z 748.534,A -85,B 0,C 180,E1 -5140.178,E2 -5140.178} C_VEL
LIN {X 0,Y 517.479,Z 738.083,A -85,B 0,C 180,E1 -5141.16,E2 -5141.16} C_VEL
LIN {X 0,Y 517.747,Z 726.413,A -85,B 0,C 180,E1 -5142.04,E2 -5142.04} C_VEL
LIN {X 0,Y 518.043,Z 714.473,A -85,B 0,C 180,E1 -5142.736,E2 -5142.736} C_VEL
LIN {X 0,Y 518.348,Z 702.147,A -85,B 0,C 180,E1 -5143.277,E2 -5143.277} C_VEL
LIN {X 0,Y 518.562,Z 688.994,A -85,B 0,C 180,E1 -5143.683,E2 -5143.683} C_VEL
LIN {X 0,Y 516.852,Z 677.999,A -85,B 0,C 180,E1 -5143.942,E2 -5143.942} C_VEL
LIN {X 0,Y 517.125,Z 662.369,A -85,B 0,C 180,E1 -5146.99,E2 -5146.99} C_VEL
LIN {X 0,Y 517.366,Z 646.341,A -85,B 0,C 180,E1 -5150.128,E2 -5150.128} C_VEL
LIN {X 0,Y 517.62,Z 630.964,A -85,B 0,C 180,E1 -5153.189,E2 -5153.189} C_VEL
LIN {X 0,Y 517.898,Z 616.913,A -85,B 0,C 180,E1 -5156.075,E2 -5156.075} C_VEL
LIN {X 0,Y 518.165,Z 601.898,A -85,B 0,C 180,E1 -5159.228,E2 -5159.228} C_VEL
LIN {X 0,Y 518.475,Z 588.392,A -85,B 0,C 180,E1 -5162.143,E2 -5162.143} C_VEL
LIN {X 0,Y 518.755,Z 574.894,A -85,B 0,C 180,E1 -5165.155,E2 -5165.155} C_VEL
LIN {X 0,Y 518.714,Z 569.699,A -85,B 0,C 180,E1 -5166.354,E2 -5166.354} C_VEL
LIN {X 0,Y 516.895,Z 560.102,A -85,B 0,C 180,E1 -5168.745,E2 -5168.745} C_VEL
LIN {X 0,Y 516.921,Z 560.098,A -85,B 0,C 180,E1 -5171.775,E2 -5171.775} C_VEL
LIN {X 0,Y 516.928,Z 560.096,A -85,B 0,C 180,E1 -5175.01,E2 -5175.01} C_VEL
LIN {X 0,Y 516.92,Z 560.097,A -85,B 0,C 180,E1 -5178.399,E2 -5178.399} C_VEL
LIN {X 0,Y 516.884,Z 560.101,A -85,B 0,C 180,E1 -5181.284,E2 -5181.284} C_VEL
LIN {X 0,Y 516.896,Z 560.1,A -85,B 0,C 180,E1 -5184.221,E2 -5184.221} C_VEL
LIN {X 0,Y 516.899,Z 560.1,A -85,B 0,C 180,E1 -5187.053,E2 -5187.053} C_VEL
LIN {X 0,Y 516.896,Z 560.102,A -85,B 0,C 180,E1 -5189.796,E2 -5189.796} C_VEL
LIN {X 0,Y 516.934,Z 560.095,A -85,B 0,C 180,E1 -5192.467,E2 -5192.467} C_VEL
LIN {X 0,Y 516.913,Z 560.097,A -85,B 0,C 180,E1 -5195.072,E2 -5195.072} C_VEL
LIN {X 0,Y 516.89,Z 560.101,A -85,B 0,C 180,E1 -5198.462,E2 -5198.462} C_VEL
LIN {X 0,Y 516.907,Z 560.099,A -85,B 0,C 180,E1 -5200.955,E2 -5200.955} C_VEL
LIN {X 0,Y 516.918,Z 560.097,A -85,B 0,C 180,E1 -5203.41,E2 -5203.41} C_VEL
LIN {X 0,Y 516.899,Z 560.099,A -85,B 0,C 180,E1 -5205.833,E2 -5205.833} C_VEL
LIN {X 0,Y 516.97,Z 560.092,A -85,B 0,C 180,E1 -5208.233,E2 -5208.233} C_VEL
LIN {X 0,Y 516.974,Z 560.089,A -85,B 0,C 180,E1 -5211.399,E2 -5211.399} C_VEL
LIN {X 0,Y 517.015,Z 560.084,A -85,B 0,C 180,E1 -5213.757,E2 -5213.757} C_VEL
LIN {X 0,Y 517.085,Z 560.077,A -85,B 0,C 180,E1 -5217.663,E2 -5217.663} C_VEL
LIN {X 0,Y 517.098,Z 560.075,A -85,B 0,C 180,E1 -5220.778,E2 -5220.778} C_VEL
LIN {X 0,Y 517.015,Z 560.085,A -85,B 0,C 180,E1 -5223.117,E2 -5223.117} C_VEL
LIN {X 0,Y 517.014,Z 560.086,A -85,B 0,C 180,E1 -5226.243,E2 -5226.243} C_VEL
LIN {X 0,Y 516.954,Z 560.093,A -85,B 0,C 180,E1 -5229.389,E2 -5229.389} C_VEL
LIN {X 0,Y 516.955,Z 560.094,A -85,B 0,C 180,E1 -5231.807,E2 -5231.807} C_VEL
LIN {X 0,Y 516.947,Z 560.094,A -85,B 0,C 180,E1 -5235.146,E2 -5235.146} C_VEL
LIN {X 0,Y 516.928,Z 560.096,A -85,B 0,C 180,E1 -5238.222,E2 -5238.222} C_VEL
LIN {X 0,Y 516.915,Z 560.098,A -85,B 0,C 180,E1 -5240.701,E2 -5240.701} C_VEL
LIN {X 0,Y 516.914,Z 560.097,A -85,B 0,C 180,E1 -5244.071,E2 -5244.071} C_VEL
LIN {X 0,Y 516.928,Z 560.097,A -85,B 0,C 180,E1 -5246.657,E2 -5246.657} C_VEL
LIN {X 0,Y 516.913,Z 560.097,A -85,B 0,C 180,E1 -5249.523,E2 -5249.523} C_VEL
LIN {X 0,Y 516.899,Z 560.101,A -85,B 0,C 180,E1 -5252.543,E2 -5252.543} C_VEL
LIN {X 0,Y 516.885,Z 560.1,A -85,B 0,C 180,E1 -5255.332,E2 -5255.332} C_VEL
LIN {X 0,Y 516.883,Z 560.101,A -85,B 0,C 180,E1 -5257.943,E2 -5257.943} C_VEL
LIN {X 0,Y 516.887,Z 560.103,A -85,B 0,C 180,E1 -5260.741,E2 -5260.741} C_VEL
LIN {X 0,Y 516.906,Z 560.099,A -85,B 0,C 180,E1 -5262.829,E2 -5262.829} C_VEL
LIN {X 0,Y 516.924,Z 560.096,A -85,B 0,C 180,E1 -5265.01,E2 -5265.01} C_VEL
LIN {X 0,Y 516.919,Z 560.097,A -85,B 0,C 180,E1 -5268.398,E2 -5268.398} C_VEL
LIN {X 0,Y 516.883,Z 560.104,A -85,B 0,C 180,E1 -5270.301,E2 -5270.301} C_VEL
LIN {X 0,Y 516.214,Z 560.186,A -85,B 0,C 180,E1 -5270.951,E2 -5270.951} C_VEL
LIN {X 0,Y 513.366,Z 560.539,A -85,B 0,C 180,E1 -5272.007,E2 -5272.007} C_VEL
LIN {X 0,Y 510.955,Z 560.841,A -85,B 0,C 180,E1 -5272.857,E2 -5272.857} C_VEL
LIN {X 0,Y 509.91,Z 560.97,A -85,B 0,C 180,E1 -5273.514,E2 -5273.514} C_VEL
LIN {X 0,Y 509.82,Z 560.981,A -85,B 0,C 180,E1 -5273.736,E2 -5273.736} C_VEL
LIN {X 0,Y 509.86,Z 560.976,A -85,B 0,C 180,E1 -5276.539,E2 -5276.539} C_VEL
LIN {X 0,Y 509.847,Z 560.978,A -85,B 0,C 180,E1 -5279.334,E2 -5279.334} C_VEL
LIN {X 0,Y 509.894,Z 560.974,A -85,B 0,C 180,E1 -5282.054,E2 -5282.054} C_VEL
LIN {X 0,Y 509.878,Z 560.974,A -85,B 0,C 180,E1 -5284.703,E2 -5284.703} C_VEL
LIN {X 0,Y 509.857,Z 560.977,A -85,B 0,C 180,E1 -5287.449,E2 -5287.449} C_VEL
LIN {X 0,Y 509.917,Z 560.968,A -85,B 0,C 180,E1 -5289.844,E2 -5289.844} C_VEL
LIN {X 0,Y 509.885,Z 560.973,A -85,B 0,C 180,E1 -5293.174,E2 -5293.174} C_VEL
LIN {X 0,Y 509.864,Z 560.975,A -85,B 0,C 180,E1 -5295.633,E2 -5295.633} C_VEL
LIN {X 0,Y 509.923,Z 560.968,A -85,B 0,C 180,E1 -5298.874,E2 -5298.874} C_VEL
LIN {X 0,Y 509.951,Z 560.966,A -85,B 0,C 180,E1 -5302.078,E2 -5302.078} C_VEL
LIN {X 0,Y 509.982,Z 560.962,A -85,B 0,C 180,E1 -5304.464,E2 -5304.464} C_VEL
LIN {X 0,Y 510.056,Z 560.954,A -85,B 0,C 180,E1 -5307.63,E2 -5307.63} C_VEL
LIN {X 0,Y 510.056,Z 560.953,A -85,B 0,C 180,E1 -5310.641,E2 -5310.641} C_VEL
LIN {X 0,Y 511.532,Z 567.054,A -85,B 0,C 180,E1 -5310.983,E2 -5310.983} C_VEL
LIN {X 0,Y 511.344,Z 579.298,A -85,B 0,C 180,E1 -5311.673,E2 -5311.673} C_VEL
LIN {X 0,Y 511.064,Z 590.246,A -85,B 0,C 180,E1 -5312.462,E2 -5312.462} C_VEL
LIN {X 0,Y 510.723,Z 600.154,A -85,B 0,C 180,E1 -5313.352,E2 -5313.352} C_VEL
LIN {X 0,Y 510.433,Z 609.075,A -85,B 0,C 180,E1 -5314.342,E2 -5314.342} C_VEL
LIN {X 0,Y 510.184,Z 616.455,A -85,B 0,C 180,E1 -5315.335,E2 -5315.335} C_VEL
LIN {X 0,Y 510.034,Z 623.956,A -85,B 0,C 180,E1 -5316.578,E2 -5316.578} C_VEL
LIN {X 0,Y 509.801,Z 630.395,A -85,B 0,C 180,E1 -5317.923,E2 -5317.923} C_VEL
LIN {X 0,Y 509.615,Z 636.051,A -85,B 0,C 180,E1 -5319.525,E2 -5319.525} C_VEL
LIN {X 0,Y 509.525,Z 638.187,A -85,B 0,C 180,E1 -5320.329,E2 -5320.329} C_VEL
LIN {X 0,Y 509.453,Z 641.123,A -85,B 0,C 180,E1 -5321.942,E2 -5321.942} C_VEL
LIN {X 0,Y 509.424,Z 641.993,A -85,B 0,C 180,E1 -5322.751,E2 -5322.751} C_VEL
LIN {X 0,Y 509.42,Z 642.464,A -85,B 0,C 180,E1 -5324.378,E2 -5324.378} C_VEL
LIN {X 0,Y 509.429,Z 642.112,A -85,B 0,C 180,E1 -5325.195,E2 -5325.195} C_VEL
LIN {X 0,Y 509.43,Z 641.318,A -85,B 0,C 180,E1 -5326.016,E2 -5326.016} C_VEL
LIN {X 0,Y 509.492,Z 640.1,A -85,B 0,C 180,E1 -5326.838,E2 -5326.838} C_VEL
LIN {X 0,Y 509.538,Z 637.955,A -85,B 0,C 180,E1 -5327.88,E2 -5327.88} C_VEL
LIN {X 0,Y 509.678,Z 633.682,A -85,B 0,C 180,E1 -5329.325,E2 -5329.325} C_VEL
LIN {X 0,Y 509.846,Z 628.65,A -85,B 0,C 180,E1 -5330.589,E2 -5330.589} C_VEL
LIN {X 0,Y 510.056,Z 622.314,A -85,B 0,C 180,E1 -5331.84,E2 -5331.84} C_VEL
LIN {X 0,Y 510.321,Z 614.157,A -85,B 0,C 180,E1 -5333.109,E2 -5333.109} C_VEL
LIN {X 0,Y 510.602,Z 605.656,A -85,B 0,C 180,E1 -5334.171,E2 -5334.171} C_VEL
LIN {X 0,Y 510.832,Z 596.697,A -85,B 0,C 180,E1 -5335.09,E2 -5335.09} C_VEL
LIN {X 0,Y 511.16,Z 587.229,A -85,B 0,C 180,E1 -5335.882,E2 -5335.882} C_VEL
LIN {X 0,Y 511.476,Z 576.674,A -85,B 0,C 180,E1 -5336.596,E2 -5336.596} C_VEL
LIN {X 0,Y 511.603,Z 567.649,A -85,B 0,C 180,E1 -5337.089,E2 -5337.089} C_VEL
LIN {X 0,Y 509.913,Z 560.97,A -85,B 0,C 180,E1 -5337.46,E2 -5337.46} C_VEL
LIN {X 0,Y 509.846,Z 560.978,A -85,B 0,C 180,E1 -5340.665,E2 -5340.665} C_VEL
LIN {X 0,Y 509.856,Z 560.976,A -85,B 0,C 180,E1 -5343.46,E2 -5343.46} C_VEL
LIN {X 0,Y 509.828,Z 560.982,A -85,B 0,C 180,E1 -5346.352,E2 -5346.352} C_VEL
LIN {X 0,Y 509.859,Z 560.977,A -85,B 0,C 180,E1 -5349.474,E2 -5349.474} C_VEL
LIN {X 0,Y 509.935,Z 560.989,A -85,B 0,C 180,E1 -5350.55,E2 -5350.55} C_VEL
LIN {X 0,Y 510.276,Z 564.808,A -85,B 0,C 180,E1 -5351.95,E2 -5351.95} C_VEL
LIN {X 0,Y 510.221,Z 573.125,A -85,B 0,C 180,E1 -5354.998,E2 -5354.998} C_VEL
LIN {X 0,Y 510.175,Z 581.595,A -85,B 0,C 180,E1 -5358.062,E2 -5358.062} C_VEL
LIN {X 0,Y 510.012,Z 588.713,A -85,B 0,C 180,E1 -5360.663,E2 -5360.663} C_VEL
LIN {X 0,Y 509.949,Z 595.232,A -85,B 0,C 180,E1 -5363.066,E2 -5363.066} C_VEL
LIN {X 0,Y 509.846,Z 603.675,A -85,B 0,C 180,E1 -5366.167,E2 -5366.167} C_VEL
LIN {X 0,Y 509.662,Z 610.651,A -85,B 0,C 180,E1 -5368.752,E2 -5368.752} C_VEL
LIN {X 0,Y 509.53,Z 618.26,A -85,B 0,C 180,E1 -5371.585,E2 -5371.585} C_VEL
LIN {X 0,Y 509.498,Z 622.014,A -85,B 0,C 180,E1 -5372.954,E2 -5372.954} C_VEL
LIN {X 0,Y 511.568,Z 634.67,A -85,B 0,C 180,E1 -5373.326,E2 -5373.326} C_VEL
LIN {X 0,Y 511.286,Z 647.35,A -85,B 0,C 180,E1 -5373.784,E2 -5373.784} C_VEL
LIN {X 0,Y 510.969,Z 660.25,A -85,B 0,C 180,E1 -5374.435,E2 -5374.435} C_VEL
LIN {X 0,Y 510.645,Z 671.514,A -85,B 0,C 180,E1 -5375.182,E2 -5375.182} C_VEL
LIN {X 0,Y 510.309,Z 681.714,A -85,B 0,C 180,E1 -5376.029,E2 -5376.029} C_VEL
LIN {X 0,Y 510.031,Z 690.118,A -85,B 0,C 180,E1 -5376.877,E2 -5376.877} C_VEL
LIN {X 0,Y 509.764,Z 698.925,A -85,B 0,C 180,E1 -5377.95,E2 -5377.95} C_VEL
LIN {X 0,Y 509.516,Z 707.247,A -85,B 0,C 180,E1 -5379.216,E2 -5379.216} C_VEL
LIN {X 0,Y 509.399,Z 712.701,A -85,B 0,C 180,E1 -5380.244,E2 -5380.244} C_VEL
LIN {X 0,Y 509.273,Z 717.988,A -85,B 0,C 180,E1 -5381.495,E2 -5381.495} C_VEL
LIN {X 0,Y 509.183,Z 722.033,A -85,B 0,C 180,E1 -5382.738,E2 -5382.738} C_VEL
LIN {X 0,Y 509.082,Z 724.964,A -85,B 0,C 180,E1 -5383.972,E2 -5383.972} C_VEL
LIN {X 0,Y 509.108,Z 726.732,A -85,B 0,C 180,E1 -5385.082,E2 -5385.082} C_VEL
LIN {X 0,Y 509.067,Z 727.809,A -85,B 0,C 180,E1 -5386.427,E2 -5386.427} C_VEL
LIN {X 0,Y 509.073,Z 727.968,A -85,B 0,C 180,E1 -5387.239,E2 -5387.239} C_VEL
LIN {X 0,Y 509.175,Z 727.285,A -85,B 0,C 180,E1 -5388.514,E2 -5388.514} C_VEL
LIN {X 0,Y 509.156,Z 725.824,A -85,B 0,C 180,E1 -5389.663,E2 -5389.663} C_VEL
LIN {X 0,Y 509.169,Z 723.348,A -85,B 0,C 180,E1 -5390.867,E2 -5390.867} C_VEL
LIN {X 0,Y 509.276,Z 719.862,A -85,B 0,C 180,E1 -5392.068,E2 -5392.068} C_VEL
LIN {X 0,Y 509.36,Z 715.296,A -85,B 0,C 180,E1 -5393.266,E2 -5393.266} C_VEL
LIN {X 0,Y 509.434,Z 709.539,A -85,B 0,C 180,E1 -5394.459,E2 -5394.459} C_VEL
LIN {X 0,Y 509.62,Z 703.665,A -85,B 0,C 180,E1 -5395.452,E2 -5395.452} C_VEL
LIN {X 0,Y 509.781,Z 696.646,A -85,B 0,C 180,E1 -5396.443,E2 -5396.443} C_VEL
LIN {X 0,Y 510.123,Z 688.16,A -85,B 0,C 180,E1 -5397.434,E2 -5397.434} C_VEL
LIN {X 0,Y 510.433,Z 677.769,A -85,B 0,C 180,E1 -5398.422,E2 -5398.422} C_VEL
LIN {X 0,Y 510.755,Z 667.361,A -85,B 0,C 180,E1 -5399.212,E2 -5399.212} C_VEL
LIN {X 0,Y 511.106,Z 655.856,A -85,B 0,C 180,E1 -5399.902,E2 -5399.902} C_VEL
LIN {X 0,Y 511.437,Z 644.041,A -85,B 0,C 180,E1 -5400.443,E2 -5400.443} C_VEL
LIN {X 0,Y 511.372,Z 632.502,A -85,B 0,C 180,E1 -5400.837,E2 -5400.837} C_VEL
LIN {X 0,Y 509.58,Z 622.281,A -85,B 0,C 180,E1 -5401.136,E2 -5401.136} C_VEL
LIN {X 0,Y 509.711,Z 613.72,A -85,B 0,C 180,E1 -5404.35,E2 -5404.35} C_VEL
LIN {X 0,Y 509.826,Z 605.041,A -85,B 0,C 180,E1 -5407.525,E2 -5407.525} C_VEL
LIN {X 0,Y 509.928,Z 598.378,A -85,B 0,C 180,E1 -5409.921,E2 -5409.921} C_VEL
LIN {X 0,Y 509.989,Z 591.61,A -85,B 0,C 180,E1 -5412.333,E2 -5412.333} C_VEL
LIN {X 0,Y 510.051,Z 582.849,A -85,B 0,C 180,E1 -5415.31,E2 -5415.31} C_VEL
LIN {X 0,Y 510.024,Z 574.486,A -85,B 0,C 180,E1 -5418.051,E2 -5418.051} C_VEL
LIN {X 0,Y 509.899,Z 565.078,A -85,B 0,C 180,E1 -5421,E2 -5421} C_VEL
LIN {X 0,Y 509.838,Z 560.981,A -85,B 0,C 180,E1 -5422.237,E2 -5422.237} C_VEL
LIN {X 0,Y 509.872,Z 560.978,A -85,B 0,C 180,E1 -5425.297,E2 -5425.297} C_VEL
LIN {X 0,Y 509.894,Z 560.974,A -85,B 0,C 180,E1 -5428.102,E2 -5428.102} C_VEL
LIN {X 0,Y 509.845,Z 560.979,A -85,B 0,C 180,E1 -5430.666,E2 -5430.666} C_VEL
LIN {X 0,Y 509.859,Z 560.978,A -85,B 0,C 180,E1 -5433.461,E2 -5433.461} C_VEL
LIN {X 0,Y 509.832,Z 560.982,A -85,B 0,C 180,E1 -5436.353,E2 -5436.353} C_VEL
LIN {X 0,Y 509.846,Z 560.98,A -85,B 0,C 180,E1 -5439.474,E2 -5439.474} C_VEL
LIN {X 0,Y 509.845,Z 560.977,A -85,B 0,C 180,E1 -5442.489,E2 -5442.489} C_VEL
LIN {X 0,Y 509.853,Z 560.978,A -85,B 0,C 180,E1 -5445.333,E2 -5445.333} C_VEL
LIN {X 0,Y 509.863,Z 560.976,A -85,B 0,C 180,E1 -5448.577,E2 -5448.577} C_VEL
LIN {X 0,Y 509.885,Z 561.138,A -85,B 0,C 180,E1 -5451.098,E2 -5451.098} C_VEL
LIN {X 0,Y 511.635,Z 569.736,A -85,B 0,C 180,E1 -5453.354,E2 -5453.354} C_VEL
LIN {X 0,Y 511.844,Z 574.227,A -85,B 0,C 180,E1 -5454.444,E2 -5454.444} C_VEL
LIN {X 0,Y 511.468,Z 586.484,A -85,B 0,C 180,E1 -5457.265,E2 -5457.265} C_VEL
LIN {X 0,Y 511.152,Z 600.373,A -85,B 0,C 180,E1 -5460.333,E2 -5460.333} C_VEL
LIN {X 0,Y 510.878,Z 612.923,A -85,B 0,C 180,E1 -5463.002,E2 -5463.002} C_VEL
LIN {X 0,Y 510.628,Z 626.567,A -85,B 0,C 180,E1 -5465.83,E2 -5465.83} C_VEL
LIN {X 0,Y 510.395,Z 641.287,A -85,B 0,C 180,E1 -5468.811,E2 -5468.811} C_VEL
LIN {X 0,Y 510.14,Z 656.848,A -85,B 0,C 180,E1 -5471.914,E2 -5471.914} C_VEL
LIN {X 0,Y 509.841,Z 673.735,A -85,B 0,C 180,E1 -5475.226,E2 -5475.226} C_VEL
LIN {X 0,Y 509.806,Z 676.979,A -85,B 0,C 180,E1 -5475.863,E2 -5475.863} C_VEL
LIN {X 0,Y 511.633,Z 690.351,A -85,B 0,C 180,E1 -5476.193,E2 -5476.193} C_VEL
LIN {X 0,Y 511.301,Z 703.881,A -85,B 0,C 180,E1 -5476.639,E2 -5476.639} C_VEL
LIN {X 0,Y 511.054,Z 715.671,A -85,B 0,C 180,E1 -5477.189,E2 -5477.189} C_VEL
LIN {X 0,Y 510.698,Z 726.78,A -85,B 0,C 180,E1 -5477.859,E2 -5477.859} C_VEL
LIN {X 0,Y 510.466,Z 737.721,A -85,B 0,C 180,E1 -5478.687,E2 -5478.687} C_VEL
LIN {X 0,Y 510.058,Z 748.377,A -85,B 0,C 180,E1 -5479.682,E2 -5479.682} C_VEL
LIN {X 0,Y 509.821,Z 756.964,A -85,B 0,C 180,E1 -5480.679,E2 -5480.679} C_VEL
LIN {X 0,Y 509.584,Z 765.239,A -85,B 0,C 180,E1 -5481.874,E2 -5481.874} C_VEL
LIN {X 0,Y 509.418,Z 771.88,A -85,B 0,C 180,E1 -5483.068,E2 -5483.068} C_VEL
LIN {X 0,Y 509.344,Z 777.952,A -85,B 0,C 180,E1 -5484.458,E2 -5484.458} C_VEL
LIN {X 0,Y 509.234,Z 781.896,A -85,B 0,C 180,E1 -5485.647,E2 -5485.647} C_VEL
LIN {X 0,Y 509.2,Z 784.808,A -85,B 0,C 180,E1 -5486.836,E2 -5486.836} C_VEL
LIN {X 0,Y 509.16,Z 786.194,A -85,B 0,C 180,E1 -5487.627,E2 -5487.627} C_VEL
LIN {X 0,Y 509.073,Z 787.786,A -85,B 0,C 180,E1 -5489.21,E2 -5489.21} C_VEL
LIN {X 0,Y 509.065,Z 788,A -85,B 0,C 180,E1 -5490.001,E2 -5490.001} C_VEL
LIN {X 0,Y 509.112,Z 787.182,A -85,B 0,C 180,E1 -5491.583,E2 -5491.583} C_VEL
LIN {X 0,Y 509.161,Z 786.195,A -85,B 0,C 180,E1 -5492.374,E2 -5492.374} C_VEL
LIN {X 0,Y 509.201,Z 784.808,A -85,B 0,C 180,E1 -5493.166,E2 -5493.166} C_VEL
LIN {X 0,Y 509.234,Z 781.893,A -85,B 0,C 180,E1 -5494.354,E2 -5494.354} C_VEL
LIN {X 0,Y 509.344,Z 777.945,A -85,B 0,C 180,E1 -5495.543,E2 -5495.543} C_VEL
LIN {X 0,Y 509.411,Z 772.277,A -85,B 0,C 180,E1 -5496.854,E2 -5496.854} C_VEL
LIN {X 0,Y 509.586,Z 765.231,A -85,B 0,C 180,E1 -5498.127,E2 -5498.127} C_VEL
LIN {X 0,Y 509.846,Z 756.955,A -85,B 0,C 180,E1 -5499.322,E2 -5499.322} C_VEL
LIN {X 0,Y 510.058,Z 748.363,A -85,B 0,C 180,E1 -5500.319,E2 -5500.319} C_VEL
LIN {X 0,Y 510.47,Z 737.712,A -85,B 0,C 180,E1 -5501.315,E2 -5501.315} C_VEL
LIN {X 0,Y 510.718,Z 726.647,A -85,B 0,C 180,E1 -5502.151,E2 -5502.151} C_VEL
LIN {X 0,Y 511.046,Z 715.668,A -85,B 0,C 180,E1 -5502.813,E2 -5502.813} C_VEL
LIN {X 0,Y 511.364,Z 703.878,A -85,B 0,C 180,E1 -5503.36,E2 -5503.36} C_VEL
LIN {X 0,Y 511.581,Z 691.247,A -85,B 0,C 180,E1 -5503.785,E2 -5503.785} C_VEL
LIN {X 0,Y 510.841,Z 684.47,A -85,B 0,C 180,E1 -5503.97,E2 -5503.97} C_VEL
LIN {X 0,Y 509.808,Z 677.121,A -85,B 0,C 180,E1 -5504.139,E2 -5504.139} C_VEL
LIN {X 0,Y 510.096,Z 660.457,A -85,B 0,C 180,E1 -5507.438,E2 -5507.438} C_VEL
LIN {X 0,Y 510.36,Z 643.979,A -85,B 0,C 180,E1 -5510.711,E2 -5510.711} C_VEL
LIN {X 0,Y 510.649,Z 628.136,A -85,B 0,C 180,E1 -5513.955,E2 -5513.955} C_VEL
LIN {X 0,Y 510.967,Z 613.591,A -85,B 0,C 180,E1 -5516.994,E2 -5516.994} C_VEL
LIN {X 0,Y 511.225,Z 599.635,A -85,B 0,C 180,E1 -5519.993,E2 -5519.993} C_VEL
LIN {X 0,Y 511.537,Z 587.187,A -85,B 0,C 180,E1 -5522.736,E2 -5522.736} C_VEL
LIN {X 0,Y 511.877,Z 573.304,A -85,B 0,C 180,E1 -5525.898,E2 -5525.898} C_VEL
LIN {X 0,Y 511.234,Z 567.816,A -85,B 0,C 180,E1 -5527.22,E2 -5527.22} C_VEL
LIN {X 0,Y 509.861,Z 560.978,A -85,B 0,C 180,E1 -5528.97,E2 -5528.97} C_VEL
LIN {X 0,Y 509.864,Z 560.978,A -85,B 0,C 180,E1 -5531.897,E2 -5531.897} C_VEL
LIN {X 0,Y 509.862,Z 560.977,A -85,B 0,C 180,E1 -5535.332,E2 -5535.332} C_VEL
LIN {X 0,Y 509.861,Z 560.976,A -85,B 0,C 180,E1 -5538.575,E2 -5538.575} C_VEL
LIN {X 0,Y 509.855,Z 560.977,A -85,B 0,C 180,E1 -5541.787,E2 -5541.787} C_VEL
LIN {X 0,Y 509.851,Z 560.978,A -85,B 0,C 180,E1 -5544.623,E2 -5544.623} C_VEL
LIN {X 0,Y 509.865,Z 560.976,A -85,B 0,C 180,E1 -5547.481,E2 -5547.481} C_VEL
LIN {X 0,Y 509.863,Z 560.976,A -85,B 0,C 180,E1 -5550.274,E2 -5550.274} C_VEL
LIN {X 0,Y 509.891,Z 560.974,A -85,B 0,C 180,E1 -5552.944,E2 -5552.944} C_VEL
LIN {X 0,Y 509.869,Z 560.976,A -85,B 0,C 180,E1 -5555.574,E2 -5555.574} C_VEL
LIN {X 0,Y 509.855,Z 560.977,A -85,B 0,C 180,E1 -5558.998,E2 -5558.998} C_VEL
LIN {X 0,Y 509.893,Z 560.972,A -85,B 0,C 180,E1 -5561.999,E2 -5561.999} C_VEL
LIN {X 0,Y 509.915,Z 560.97,A -85,B 0,C 180,E1 -5564.819,E2 -5564.819} C_VEL
LIN {X 0,Y 509.905,Z 560.971,A -85,B 0,C 180,E1 -5568.124,E2 -5568.124} C_VEL
LIN {X 0,Y 509.92,Z 560.967,A -85,B 0,C 180,E1 -5571.28,E2 -5571.28} C_VEL
LIN {X 0,Y 509.983,Z 560.96,A -85,B 0,C 180,E1 -5573.67,E2 -5573.67} C_VEL
LIN {X 0,Y 510.056,Z 560.952,A -85,B 0,C 180,E1 -5577.631,E2 -5577.631} C_VEL
LIN {X 0,Y 510.068,Z 560.951,A -85,B 0,C 180,E1 -5580.789,E2 -5580.789} C_VEL
LIN {X 0,Y 509.957,Z 560.964,A -85,B 0,C 180,E1 -5583.16,E2 -5583.16} C_VEL
LIN {X 0,Y 509.982,Z 560.961,A -85,B 0,C 180,E1 -5586.329,E2 -5586.329} C_VEL
LIN {X 0,Y 509.918,Z 560.969,A -85,B 0,C 180,E1 -5588.72,E2 -5588.72} C_VEL
LIN {X 0,Y 509.907,Z 560.971,A -85,B 0,C 180,E1 -5591.931,E2 -5591.931} C_VEL
LIN {X 0,Y 509.897,Z 560.972,A -85,B 0,C 180,E1 -5595.241,E2 -5595.241} C_VEL
LIN {X 0,Y 509.891,Z 560.972,A -85,B 0,C 180,E1 -5598,E2 -5598} C_VEL
LIN {X 0,Y 509.853,Z 560.978,A -85,B 0,C 180,E1 -5601.001,E2 -5601.001} C_VEL
LIN {X 0,Y 509.839,Z 560.979,A -85,B 0,C 180,E1 -5603.563,E2 -5603.563} C_VEL
LIN {X 0,Y 509.914,Z 560.97,A -85,B 0,C 180,E1 -5606.378,E2 -5606.378} C_VEL
LIN {X 0,Y 509.879,Z 560.974,A -85,B 0,C 180,E1 -5608.844,E2 -5608.844} C_VEL
LIN {X 0,Y 509.823,Z 560.981,A -85,B 0,C 180,E1 -5611.59,E2 -5611.59} C_VEL
LIN {X 0,Y 509.856,Z 560.977,A -85,B 0,C 180,E1 -5614.413,E2 -5614.413} C_VEL
LIN {X 0,Y 509.821,Z 560.981,A -85,B 0,C 180,E1 -5617.34,E2 -5617.34} C_VEL
LIN {X 0,Y 509.84,Z 560.979,A -85,B 0,C 180,E1 -5620.382,E2 -5620.382} C_VEL
LIN {X 0,Y 509.841,Z 560.98,A -85,B 0,C 180,E1 -5623.064,E2 -5623.064} C_VEL
LIN {X 0,Y 509.832,Z 560.981,A -85,B 0,C 180,E1 -5625.792,E2 -5625.792} C_VEL
LIN {X 0,Y 509.86,Z 560.976,A -85,B 0,C 180,E1 -5628.574,E2 -5628.574} C_VEL
LIN {X 0,Y 509.853,Z 560.977,A -85,B 0,C 180,E1 -5631.786,E2 -5631.786} C_VEL
LIN {X 0,Y 509.82,Z 560.981,A -85,B 0,C 180,E1 -5633.736,E2 -5633.736} C_VEL
LIN {X 0,Y 509.152,Z 561.065,A -85,B 0,C 180,E1 -5634.396,E2 -5634.396} C_VEL
LIN {X 0,Y 506.339,Z 561.415,A -85,B 0,C 180,E1 -5635.468,E2 -5635.468} C_VEL
LIN {X 0,Y 503.953,Z 561.714,A -85,B 0,C 180,E1 -5636.331,E2 -5636.331} C_VEL
LIN {X 0,Y 502.907,Z 561.844,A -85,B 0,C 180,E1 -5636.998,E2 -5636.998} C_VEL
LIN {X 0,Y 502.81,Z 561.854,A -85,B 0,C 180,E1 -5637.223,E2 -5637.223} C_VEL
LIN {X 0,Y 502.815,Z 561.854,A -85,B 0,C 180,E1 -5640.064,E2 -5640.064} C_VEL
LIN {X 0,Y 502.834,Z 561.852,A -85,B 0,C 180,E1 -5642.533,E2 -5642.533} C_VEL
LIN {X 0,Y 502.829,Z 561.852,A -85,B 0,C 180,E1 -5645.298,E2 -5645.298} C_VEL
LIN {X 0,Y 502.794,Z 561.857,A -85,B 0,C 180,E1 -5647.826,E2 -5647.826} C_VEL
LIN {X 0,Y 502.826,Z 561.853,A -85,B 0,C 180,E1 -5650.4,E2 -5650.4} C_VEL
LIN {X 0,Y 502.834,Z 561.851,A -85,B 0,C 180,E1 -5652.931,E2 -5652.931} C_VEL
LIN {X 0,Y 502.845,Z 561.849,A -85,B 0,C 180,E1 -5655.429,E2 -5655.429} C_VEL
LIN {X 0,Y 502.893,Z 561.844,A -85,B 0,C 180,E1 -5658.717,E2 -5658.717} C_VEL
LIN {X 0,Y 502.901,Z 561.844,A -85,B 0,C 180,E1 -5661.966,E2 -5661.966} C_VEL
LIN {X 0,Y 502.938,Z 561.839,A -85,B 0,C 180,E1 -5664.386,E2 -5664.386} C_VEL
LIN {X 0,Y 503.025,Z 561.83,A -85,B 0,C 180,E1 -5667.597,E2 -5667.597} C_VEL
LIN {X 0,Y 503.023,Z 561.829,A -85,B 0,C 180,E1 -5670.45,E2 -5670.45} C_VEL
LIN {X 0,Y 504.583,Z 568.022,A -85,B 0,C 180,E1 -5670.797,E2 -5670.797} C_VEL
LIN {X 0,Y 504.528,Z 578.648,A -85,B 0,C 180,E1 -5671.396,E2 -5671.396} C_VEL
LIN {X 0,Y 504.197,Z 589.908,A -85,B 0,C 180,E1 -5672.196,E2 -5672.196} C_VEL
LIN {X 0,Y 503.829,Z 600.08,A -85,B 0,C 180,E1 -5673.098,E2 -5673.098} C_VEL
LIN {X 0,Y 503.604,Z 608.373,A -85,B 0,C 180,E1 -5674,E2 -5674} C_VEL
LIN {X 0,Y 503.284,Z 616.074,A -85,B 0,C 180,E1 -5675.006,E2 -5675.006} C_VEL
LIN {X 0,Y 503.091,Z 623.561,A -85,B 0,C 180,E1 -5676.214,E2 -5676.214} C_VEL
LIN {X 0,Y 502.926,Z 628.712,A -85,B 0,C 180,E1 -5677.224,E2 -5677.224} C_VEL
LIN {X 0,Y 502.742,Z 633.708,A -85,B 0,C 180,E1 -5678.44,E2 -5678.44} C_VEL
LIN {X 0,Y 502.583,Z 637.599,A -85,B 0,C 180,E1 -5679.659,E2 -5679.659} C_VEL
LIN {X 0,Y 502.496,Z 639.62,A -85,B 0,C 180,E1 -5680.475,E2 -5680.475} C_VEL
LIN {X 0,Y 502.459,Z 641.881,A -85,B 0,C 180,E1 -5681.735,E2 -5681.735} C_VEL
LIN {X 0,Y 502.406,Z 643.13,A -85,B 0,C 180,E1 -5682.933,E2 -5682.933} C_VEL
LIN {X 0,Y 502.414,Z 643.432,A -85,B 0,C 180,E1 -5684.583,E2 -5684.583} C_VEL
LIN {X 0,Y 502.424,Z 642.974,A -85,B 0,C 180,E1 -5685.412,E2 -5685.412} C_VEL
LIN {X 0,Y 502.421,Z 642.08,A -85,B 0,C 180,E1 -5686.245,E2 -5686.245} C_VEL
LIN {X 0,Y 502.484,Z 640.765,A -85,B 0,C 180,E1 -5687.08,E2 -5687.08} C_VEL
LIN {X 0,Y 502.577,Z 638.047,A -85,B 0,C 180,E1 -5688.296,E2 -5688.296} C_VEL
LIN {X 0,Y 502.712,Z 634.003,A -85,B 0,C 180,E1 -5689.603,E2 -5689.603} C_VEL
LIN {X 0,Y 502.938,Z 627.804,A -85,B 0,C 180,E1 -5691.088,E2 -5691.088} C_VEL
LIN {X 0,Y 503.184,Z 621.132,A -85,B 0,C 180,E1 -5692.326,E2 -5692.326} C_VEL
LIN {X 0,Y 503.495,Z 613.68,A -85,B 0,C 180,E1 -5693.441,E2 -5693.441} C_VEL
LIN {X 0,Y 503.766,Z 604.826,A -85,B 0,C 180,E1 -5694.521,E2 -5694.521} C_VEL
LIN {X 0,Y 504.068,Z 594.751,A -85,B 0,C 180,E1 -5695.51,E2 -5695.51} C_VEL
LIN {X 0,Y 504.472,Z 583.9,A -85,B 0,C 180,E1 -5696.362,E2 -5696.362} C_VEL
LIN {X 0,Y 504.69,Z 572.006,A -85,B 0,C 180,E1 -5697.097,E2 -5697.097} C_VEL
LIN {X 0,Y 504.46,Z 567.636,A -85,B 0,C 180,E1 -5697.333,E2 -5697.333} C_VEL
LIN {X 0,Y 502.851,Z 561.85,A -85,B 0,C 180,E1 -5697.662,E2 -5697.662} C_VEL
LIN {X 0,Y 502.815,Z 561.856,A -85,B 0,C 180,E1 -5700.21,E2 -5700.21} C_VEL
LIN {X 0,Y 502.826,Z 561.853,A -85,B 0,C 180,E1 -5703.031,E2 -5703.031} C_VEL
LIN {X 0,Y 502.775,Z 561.859,A -85,B 0,C 180,E1 -5705.95,E2 -5705.95} C_VEL
LIN {X 0,Y 502.815,Z 561.855,A -85,B 0,C 180,E1 -5708.973,E2 -5708.973} C_VEL
LIN {X 0,Y 502.9,Z 561.969,A -85,B 0,C 180,E1 -5710.462,E2 -5710.462} C_VEL
LIN {X 0,Y 503.308,Z 566.846,A -85,B 0,C 180,E1 -5712.263,E2 -5712.263} C_VEL
LIN {X 0,Y 503.228,Z 575.36,A -85,B 0,C 180,E1 -5715.417,E2 -5715.417} C_VEL
LIN {X 0,Y 503.128,Z 583.635,A -85,B 0,C 180,E1 -5718.432,E2 -5718.432} C_VEL
LIN {X 0,Y 502.982,Z 590.769,A -85,B 0,C 180,E1 -5721.041,E2 -5721.041} C_VEL
LIN {X 0,Y 502.877,Z 598.927,A -85,B 0,C 180,E1 -5724.058,E2 -5724.058} C_VEL
LIN {X 0,Y 502.742,Z 606.894,A -85,B 0,C 180,E1 -5727.007,E2 -5727.007} C_VEL
LIN {X 0,Y 502.582,Z 615.254,A -85,B 0,C 180,E1 -5730.109,E2 -5730.109} C_VEL
LIN {X 0,Y 502.477,Z 622.579,A -85,B 0,C 180,E1 -5732.769,E2 -5732.769} C_VEL
LIN {X 0,Y 504.69,Z 635.166,A -85,B 0,C 180,E1 -5733.146,E2 -5733.146} C_VEL
LIN {X 0,Y 504.365,Z 648.29,A -85,B 0,C 180,E1 -5733.631,E2 -5733.631} C_VEL
LIN {X 0,Y 504.029,Z 660.781,A -85,B 0,C 180,E1 -5734.279,E2 -5734.279} C_VEL
LIN {X 0,Y 503.673,Z 672.734,A -85,B 0,C 180,E1 -5735.088,E2 -5735.088} C_VEL
LIN {X 0,Y 503.324,Z 683.381,A -85,B 0,C 180,E1 -5736.004,E2 -5736.004} C_VEL
LIN {X 0,Y 503.019,Z 692.502,A -85,B 0,C 180,E1 -5736.971,E2 -5736.971} C_VEL
LIN {X 0,Y 502.702,Z 700.794,A -85,B 0,C 180,E1 -5738.039,E2 -5738.039} C_VEL
LIN {X 0,Y 502.462,Z 708.751,A -85,B 0,C 180,E1 -5739.319,E2 -5739.319} C_VEL
LIN {X 0,Y 502.317,Z 714.094,A -85,B 0,C 180,E1 -5740.38,E2 -5740.38} C_VEL
LIN {X 0,Y 502.211,Z 719.187,A -85,B 0,C 180,E1 -5741.648,E2 -5741.648} C_VEL
LIN {X 0,Y 502.098,Z 723.052,A -85,B 0,C 180,E1 -5742.906,E2 -5742.906} C_VEL
LIN {X 0,Y 502.022,Z 725.034,A -85,B 0,C 180,E1 -5743.741,E2 -5743.741} C_VEL
LIN {X 0,Y 502.045,Z 727.095,A -85,B 0,C 180,E1 -5744.993,E2 -5744.993} C_VEL
LIN {X 0,Y 501.992,Z 728.182,A -85,B 0,C 180,E1 -5746.232,E2 -5746.232} C_VEL
LIN {X 0,Y 501.98,Z 728.42,A -85,B 0,C 180,E1 -5747.056,E2 -5747.056} C_VEL
LIN {X 0,Y 502.104,Z 727.549,A -85,B 0,C 180,E1 -5748.7,E2 -5748.7} C_VEL
LIN {X 0,Y 502.1,Z 726.558,A -85,B 0,C 180,E1 -5749.516,E2 -5749.516} C_VEL
LIN {X 0,Y 502.042,Z 725.099,A -85,B 0,C 180,E1 -5750.33,E2 -5750.33} C_VEL
LIN {X 0,Y 502.208,Z 720.908,A -85,B 0,C 180,E1 -5751.956,E2 -5751.956} C_VEL
LIN {X 0,Y 502.277,Z 716.519,A -85,B 0,C 180,E1 -5753.17,E2 -5753.17} C_VEL
LIN {X 0,Y 502.405,Z 710.924,A -85,B 0,C 180,E1 -5754.381,E2 -5754.381} C_VEL
LIN {X 0,Y 502.593,Z 703.954,A -85,B 0,C 180,E1 -5755.589,E2 -5755.589} C_VEL
LIN {X 0,Y 502.855,Z 695.321,A -85,B 0,C 180,E1 -5756.796,E2 -5756.796} C_VEL
LIN {X 0,Y 503.212,Z 686.439,A -85,B 0,C 180,E1 -5757.799,E2 -5757.799} C_VEL
LIN {X 0,Y 503.56,Z 675.405,A -85,B 0,C 180,E1 -5758.801,E2 -5758.801} C_VEL
LIN {X 0,Y 503.941,Z 664.36,A -85,B 0,C 180,E1 -5759.601,E2 -5759.601} C_VEL
LIN {X 0,Y 504.303,Z 651.792,A -85,B 0,C 180,E1 -5760.3,E2 -5760.3} C_VEL
LIN {X 0,Y 504.605,Z 639.753,A -85,B 0,C 180,E1 -5760.798,E2 -5760.798} C_VEL
LIN {X 0,Y 504.443,Z 632.938,A -85,B 0,C 180,E1 -5761.023,E2 -5761.023} C_VEL
LIN {X 0,Y 502.53,Z 622.778,A -85,B 0,C 180,E1 -5761.328,E2 -5761.328} C_VEL
LIN {X 0,Y 502.754,Z 613.418,A -85,B 0,C 180,E1 -5764.812,E2 -5764.812} C_VEL
LIN {X 0,Y 502.842,Z 603.503,A -85,B 0,C 180,E1 -5768.439,E2 -5768.439} C_VEL
LIN {X 0,Y 502.951,Z 595.635,A -85,B 0,C 180,E1 -5771.282,E2 -5771.282} C_VEL
LIN {X 0,Y 503.007,Z 588.551,A -85,B 0,C 180,E1 -5773.741,E2 -5773.741} C_VEL
LIN {X 0,Y 503.009,Z 579.893,A -85,B 0,C 180,E1 -5776.644,E2 -5776.644} C_VEL
LIN {X 0,Y 502.954,Z 570.761,A -85,B 0,C 180,E1 -5779.595,E2 -5779.595} C_VEL
LIN {X 0,Y 502.798,Z 561.858,A -85,B 0,C 180,E1 -5782.363,E2 -5782.363} C_VEL
LIN {X 0,Y 502.835,Z 561.855,A -85,B 0,C 180,E1 -5785.676,E2 -5785.676} C_VEL
LIN {X 0,Y 502.837,Z 561.852,A -85,B 0,C 180,E1 -5788.373,E2 -5788.373} C_VEL
LIN {X 0,Y 502.792,Z 561.858,A -85,B 0,C 180,E1 -5791.501,E2 -5791.501} C_VEL
LIN {X 0,Y 502.802,Z 561.858,A -85,B 0,C 180,E1 -5794.446,E2 -5794.446} C_VEL
LIN {X 0,Y 502.779,Z 561.858,A -85,B 0,C 180,E1 -5797.18,E2 -5797.18} C_VEL
LIN {X 0,Y 502.817,Z 561.853,A -85,B 0,C 180,E1 -5800.013,E2 -5800.013} C_VEL
LIN {X 0,Y 502.825,Z 561.85,A -85,B 0,C 180,E1 -5802.204,E2 -5802.204} C_VEL
LIN {X 0,Y 502.797,Z 561.857,A -85,B 0,C 180,E1 -5805.469,E2 -5805.469} C_VEL
LIN {X 0,Y 502.827,Z 561.854,A -85,B 0,C 180,E1 -5807.865,E2 -5807.865} C_VEL
LIN {X 0,Y 502.856,Z 561.89,A -85,B 0,C 180,E1 -5810.772,E2 -5810.772} C_VEL
LIN {X 0,Y 504.883,Z 572.416,A -85,B 0,C 180,E1 -5813.579,E2 -5813.579} C_VEL
LIN {X 0,Y 504.743,Z 581.225,A -85,B 0,C 180,E1 -5815.69,E2 -5815.69} C_VEL
LIN {X 0,Y 504.346,Z 593.821,A -85,B 0,C 180,E1 -5818.586,E2 -5818.586} C_VEL
LIN {X 0,Y 504.009,Z 607.927,A -85,B 0,C 180,E1 -5821.7,E2 -5821.7} C_VEL
LIN {X 0,Y 503.68,Z 622.373,A -85,B 0,C 180,E1 -5824.778,E2 -5824.778} C_VEL
LIN {X 0,Y 503.398,Z 635.413,A -85,B 0,C 180,E1 -5827.489,E2 -5827.489} C_VEL
LIN {X 0,Y 503.174,Z 649.757,A -85,B 0,C 180,E1 -5830.415,E2 -5830.415} C_VEL
LIN {X 0,Y 502.903,Z 664.344,A -85,B 0,C 180,E1 -5833.353,E2 -5833.353} C_VEL
LIN {X 0,Y 502.727,Z 675.904,A -85,B 0,C 180,E1 -5835.659,E2 -5835.659} C_VEL
LIN {X 0,Y 504.048,Z 686.172,A -85,B 0,C 180,E1 -5835.9,E2 -5835.9} C_VEL
LIN {X 0,Y 504.658,Z 692.052,A -85,B 0,C 180,E1 -5836.075,E2 -5836.075} C_VEL
LIN {X 0,Y 504.293,Z 705.189,A -85,B 0,C 180,E1 -5836.553,E2 -5836.553} C_VEL
LIN {X 0,Y 503.954,Z 717.861,A -85,B 0,C 180,E1 -5837.192,E2 -5837.192} C_VEL
LIN {X 0,Y 503.631,Z 729.012,A -85,B 0,C 180,E1 -5837.918,E2 -5837.918} C_VEL
LIN {X 0,Y 503.281,Z 740.104,A -85,B 0,C 180,E1 -5838.829,E2 -5838.829} C_VEL
LIN {X 0,Y 502.946,Z 749.159,A -85,B 0,C 180,E1 -5839.738,E2 -5839.738} C_VEL
LIN {X 0,Y 502.697,Z 759.032,A -85,B 0,C 180,E1 -5840.952,E2 -5840.952} C_VEL
LIN {X 0,Y 502.445,Z 766.906,A -85,B 0,C 180,E1 -5842.162,E2 -5842.162} C_VEL
LIN {X 0,Y 502.255,Z 774.173,A -85,B 0,C 180,E1 -5843.573,E2 -5843.573} C_VEL
LIN {X 0,Y 502.186,Z 779.022,A -85,B 0,C 180,E1 -5844.782,E2 -5844.782} C_VEL
LIN {X 0,Y 502.15,Z 782.731,A -85,B 0,C 180,E1 -5845.988,E2 -5845.988} C_VEL
LIN {X 0,Y 502.121,Z 784.636,A -85,B 0,C 180,E1 -5846.791,E2 -5846.791} C_VEL
LIN {X 0,Y 502.065,Z 786.056,A -85,B 0,C 180,E1 -5847.594,E2 -5847.594} C_VEL
LIN {X 0,Y 502.035,Z 787.067,A -85,B 0,C 180,E1 -5848.396,E2 -5848.396} C_VEL
LIN {X 0,Y 501.98,Z 787.899,A -85,B 0,C 180,E1 -5850.001,E2 -5850.001} C_VEL
LIN {X 0,Y 502.035,Z 787.068,A -85,B 0,C 180,E1 -5851.605,E2 -5851.605} C_VEL
LIN {X 0,Y 502.065,Z 786.057,A -85,B 0,C 180,E1 -5852.408,E2 -5852.408} C_VEL
LIN {X 0,Y 502.121,Z 784.637,A -85,B 0,C 180,E1 -5853.21,E2 -5853.21} C_VEL
LIN {X 0,Y 502.126,Z 781.623,A -85,B 0,C 180,E1 -5854.416,E2 -5854.416} C_VEL
LIN {X 0,Y 502.26,Z 777.557,A -85,B 0,C 180,E1 -5855.622,E2 -5855.622} C_VEL
LIN {X 0,Y 502.337,Z 771.391,A -85,B 0,C 180,E1 -5857.012,E2 -5857.012} C_VEL
LIN {X 0,Y 502.516,Z 764.453,A -85,B 0,C 180,E1 -5858.243,E2 -5858.243} C_VEL
LIN {X 0,Y 502.791,Z 756.009,A -85,B 0,C 180,E1 -5859.454,E2 -5859.454} C_VEL
LIN {X 0,Y 503.039,Z 747.35,A -85,B 0,C 180,E1 -5860.465,E2 -5860.465} C_VEL
LIN {X 0,Y 503.423,Z 736.693,A -85,B 0,C 180,E1 -5861.475,E2 -5861.475} C_VEL
LIN {X 0,Y 503.711,Z 725.631,A -85,B 0,C 180,E1 -5862.323,E2 -5862.323} C_VEL
LIN {X 0,Y 504.048,Z 714.65,A -85,B 0,C 180,E1 -5862.994,E2 -5862.994} C_VEL
LIN {X 0,Y 504.421,Z 702.865,A -85,B 0,C 180,E1 -5863.548,E2 -5863.548} C_VEL
LIN {X 0,Y 504.583,Z 689.763,A -85,B 0,C 180,E1 -5863.993,E2 -5863.993} C_VEL
LIN {X 0,Y 502.851,Z 677.858,A -85,B 0,C 180,E1 -5864.301,E2 -5864.301} C_VEL
LIN {X 0,Y 502.751,Z 675.973,A -85,B 0,C 180,E1 -5864.367,E2 -5864.367} C_VEL
LIN {X 0,Y 503.013,Z 659.565,A -85,B 0,C 180,E1 -5867.692,E2 -5867.692} C_VEL
LIN {X 0,Y 503.292,Z 643.497,A -85,B 0,C 180,E1 -5870.932,E2 -5870.932} C_VEL
LIN {X 0,Y 503.597,Z 628.342,A -85,B 0,C 180,E1 -5874.092,E2 -5874.092} C_VEL
LIN {X 0,Y 503.938,Z 614.423,A -85,B 0,C 180,E1 -5877.054,E2 -5877.054} C_VEL
LIN {X 0,Y 504.269,Z 599.91,A -85,B 0,C 180,E1 -5880.22,E2 -5880.22} C_VEL
LIN {X 0,Y 504.578,Z 587.907,A -85,B 0,C 180,E1 -5882.903,E2 -5882.903} C_VEL
LIN {X 0,Y 504.958,Z 573.779,A -85,B 0,C 180,E1 -5886.172,E2 -5886.172} C_VEL
LIN {X 0,Y 503.846,Z 567.038,A -85,B 0,C 180,E1 -5887.861,E2 -5887.861} C_VEL
LIN {X 0,Y 502.811,Z 561.855,A -85,B 0,C 180,E1 -5889.234,E2 -5889.234} C_VEL
LIN {X 0,Y 502.808,Z 561.857,A -85,B 0,C 180,E1 -5892.199,E2 -5892.199} C_VEL
LIN {X 0,Y 502.806,Z 561.857,A -85,B 0,C 180,E1 -5895.468,E2 -5895.468} C_VEL
LIN {X 0,Y 502.825,Z 561.854,A -85,B 0,C 180,E1 -5898.934,E2 -5898.934} C_VEL
LIN {X 0,Y 502.798,Z 561.856,A -85,B 0,C 180,E1 -5902.046,E2 -5902.046} C_VEL
LIN {X 0,Y 502.815,Z 561.854,A -85,B 0,C 180,E1 -5905.035,E2 -5905.035} C_VEL
LIN {X 0,Y 502.788,Z 561.857,A -85,B 0,C 180,E1 -5907.915,E2 -5907.915} C_VEL
LIN {X 0,Y 502.829,Z 561.854,A -85,B 0,C 180,E1 -5910.712,E2 -5910.712} C_VEL
LIN {X 0,Y 502.867,Z 561.847,A -85,B 0,C 180,E1 -5913.439,E2 -5913.439} C_VEL
LIN {X 0,Y 502.79,Z 561.857,A -85,B 0,C 180,E1 -5916.086,E2 -5916.086} C_VEL
LIN {X 0,Y 502.788,Z 561.858,A -85,B 0,C 180,E1 -5918.689,E2 -5918.689} C_VEL
LIN {X 0,Y 502.834,Z 561.851,A -85,B 0,C 180,E1 -5921.248,E2 -5921.248} C_VEL
LIN {X 0,Y 502.827,Z 561.853,A -85,B 0,C 180,E1 -5923.767,E2 -5923.767} C_VEL
LIN {X 0,Y 502.835,Z 561.852,A -85,B 0,C 180,E1 -5926.254,E2 -5926.254} C_VEL
LIN {X 0,Y 502.881,Z 561.845,A -85,B 0,C 180,E1 -5928.717,E2 -5928.717} C_VEL
LIN {X 0,Y 502.906,Z 561.844,A -85,B 0,C 180,E1 -5931.966,E2 -5931.966} C_VEL
LIN {X 0,Y 502.943,Z 561.839,A -85,B 0,C 180,E1 -5934.386,E2 -5934.386} C_VEL
LIN {X 0,Y 503.026,Z 561.827,A -85,B 0,C 180,E1 -5937.597,E2 -5937.597} C_VEL
LIN {X 0,Y 503.031,Z 561.828,A -85,B 0,C 180,E1 -5940,E2 -5940} C_VEL
LIN {X 0,Y 503.027,Z 561.829,A -85,B 0,C 180,E1 -5942.402,E2 -5942.402} C_VEL
LIN {X 0,Y 502.942,Z 561.837,A -85,B 0,C 180,E1 -5945.613,E2 -5945.613} C_VEL
LIN {X 0,Y 502.905,Z 561.843,A -85,B 0,C 180,E1 -5948.033,E2 -5948.033} C_VEL
LIN {X 0,Y 502.88,Z 561.845,A -85,B 0,C 180,E1 -5951.283,E2 -5951.283} C_VEL
LIN {X 0,Y 502.848,Z 561.85,A -85,B 0,C 180,E1 -5954.57,E2 -5954.57} C_VEL
LIN {X 0,Y 502.865,Z 561.848,A -85,B 0,C 180,E1 -5957.906,E2 -5957.906} C_VEL
LIN {X 0,Y 502.831,Z 561.852,A -85,B 0,C 180,E1 -5960.536,E2 -5960.536} C_VEL
LIN {X 0,Y 502.8,Z 561.856,A -85,B 0,C 180,E1 -5963.04,E2 -5963.04} C_VEL
LIN {X 0,Y 502.843,Z 561.85,A -85,B 0,C 180,E1 -5965.675,E2 -5965.675} C_VEL
LIN {X 0,Y 502.842,Z 561.851,A -85,B 0,C 180,E1 -5968.372,E2 -5968.372} C_VEL
LIN {X 0,Y 502.795,Z 561.856,A -85,B 0,C 180,E1 -5971.498,E2 -5971.498} C_VEL
LIN {X 0,Y 502.808,Z 561.855,A -85,B 0,C 180,E1 -5974.444,E2 -5974.444} C_VEL
LIN {X 0,Y 502.783,Z 561.859,A -85,B 0,C 180,E1 -5977.178,E2 -5977.178} C_VEL
LIN {X 0,Y 502.79,Z 561.858,A -85,B 0,C 180,E1 -5980.015,E2 -5980.015} C_VEL
LIN {X 0,Y 502.804,Z 561.857,A -85,B 0,C 180,E1 -5982.199,E2 -5982.199} C_VEL
LIN {X 0,Y 502.802,Z 561.855,A -85,B 0,C 180,E1 -5985.468,E2 -5985.468} C_VEL
LIN {X 0,Y 502.831,Z 561.852,A -85,B 0,C 180,E1 -5987.864,E2 -5987.864} C_VEL
LIN {X 0,Y 502.804,Z 561.856,A -85,B 0,C 180,E1 -5991.024,E2 -5991.024} C_VEL
LIN {X 0,Y 502.775,Z 561.859,A -85,B 0,C 180,E1 -5994.168,E2 -5994.168} C_VEL
LIN {X 0,Y 502.81,Z 561.854,A -85,B 0,C 180,E1 -5997.223,E2 -5997.223} C_VEL
LIN {X 0,Y 502.11,Z 561.941,A -85,B 0,C 180,E1 -5997.892,E2 -5997.892} C_VEL
LIN {X 0,Y 499.245,Z 562.298,A -85,B 0,C 180,E1 -5998.978,E2 -5998.978} C_VEL
LIN {X 0,Y 496.849,Z 562.598,A -85,B 0,C 180,E1 -5999.853,E2 -5999.853} C_VEL
LIN {X 0,Y 495.832,Z 562.725,A -85,B 0,C 180,E1 -6000.528,E2 -6000.528} C_VEL
LIN {X 0,Y 495.754,Z 562.731,A -85,B 0,C 180,E1 -6000.757,E2 -6000.757} C_VEL
LIN {X 0,Y 495.791,Z 562.727,A -85,B 0,C 180,E1 -6003.932,E2 -6003.932} C_VEL
LIN {X 0,Y 495.759,Z 562.732,A -85,B 0,C 180,E1 -6007.139,E2 -6007.139} C_VEL
LIN {X 0,Y 495.772,Z 562.732,A -85,B 0,C 180,E1 -6010.109,E2 -6010.109} C_VEL
LIN {X 0,Y 495.787,Z 562.73,A -85,B 0,C 180,E1 -6012.681,E2 -6012.681} C_VEL
LIN {X 0,Y 495.79,Z 562.728,A -85,B 0,C 180,E1 -6015.217,E2 -6015.217} C_VEL
LIN {X 0,Y 495.868,Z 562.72,A -85,B 0,C 180,E1 -6018.555,E2 -6018.555} C_VEL
LIN {X 0,Y 495.872,Z 562.719,A -85,B 0,C 180,E1 -6021.851,E2 -6021.851} C_VEL
LIN {X 0,Y 495.896,Z 562.717,A -85,B 0,C 180,E1 -6024.306,E2 -6024.306} C_VEL
LIN {X 0,Y 495.994,Z 562.706,A -85,B 0,C 180,E1 -6027.563,E2 -6027.563} C_VEL
LIN {X 0,Y 495.993,Z 562.705,A -85,B 0,C 180,E1 -6030.253,E2 -6030.253} C_VEL
LIN {X 0,Y 497.86,Z 570.659,A -85,B 0,C 180,E1 -6030.707,E2 -6030.707} C_VEL
LIN {X 0,Y 497.573,Z 582.59,A -85,B 0,C 180,E1 -6031.416,E2 -6031.416} C_VEL
LIN {X 0,Y 497.276,Z 593.266,A -85,B 0,C 180,E1 -6032.227,E2 -6032.227} C_VEL
LIN {X 0,Y 496.959,Z 601.984,A -85,B 0,C 180,E1 -6033.039,E2 -6033.039} C_VEL
LIN {X 0,Y 496.633,Z 610.942,A -85,B 0,C 180,E1 -6034.057,E2 -6034.057} C_VEL
LIN {X 0,Y 496.269,Z 619.686,A -85,B 0,C 180,E1 -6035.281,E2 -6035.281} C_VEL
LIN {X 0,Y 496.103,Z 626.702,A -85,B 0,C 180,E1 -6036.507,E2 -6036.507} C_VEL
LIN {X 0,Y 495.828,Z 632.346,A -85,B 0,C 180,E1 -6037.738,E2 -6037.738} C_VEL
LIN {X 0,Y 495.669,Z 636.78,A -85,B 0,C 180,E1 -6038.972,E2 -6038.972} C_VEL
LIN {X 0,Y 495.553,Z 639.125,A -85,B 0,C 180,E1 -6039.798,E2 -6039.798} C_VEL
LIN {X 0,Y 495.471,Z 641.05,A -85,B 0,C 180,E1 -6040.625,E2 -6040.625} C_VEL
LIN {X 0,Y 495.437,Z 643.046,A -85,B 0,C 180,E1 -6041.822,E2 -6041.822} C_VEL
LIN {X 0,Y 495.372,Z 644.257,A -85,B 0,C 180,E1 -6043.119,E2 -6043.119} C_VEL
LIN {X 0,Y 495.39,Z 644.526,A -85,B 0,C 180,E1 -6043.955,E2 -6043.955} C_VEL
LIN {X 0,Y 495.418,Z 644.101,A -85,B 0,C 180,E1 -6045.282,E2 -6045.282} C_VEL
LIN {X 0,Y 495.435,Z 642.819,A -85,B 0,C 180,E1 -6046.481,E2 -6046.481} C_VEL
LIN {X 0,Y 495.478,Z 641.415,A -85,B 0,C 180,E1 -6047.329,E2 -6047.329} C_VEL
LIN {X 0,Y 495.628,Z 638.417,A -85,B 0,C 180,E1 -6048.605,E2 -6048.605} C_VEL
LIN {X 0,Y 495.759,Z 634.28,A -85,B 0,C 180,E1 -6049.89,E2 -6049.89} C_VEL
LIN {X 0,Y 496.023,Z 627.82,A -85,B 0,C 180,E1 -6051.397,E2 -6051.397} C_VEL
LIN {X 0,Y 496.24,Z 621.936,A -85,B 0,C 180,E1 -6052.481,E2 -6052.481} C_VEL
LIN {X 0,Y 496.566,Z 614.762,A -85,B 0,C 180,E1 -6053.566,E2 -6053.566} C_VEL
LIN {X 0,Y 496.876,Z 605.941,A -85,B 0,C 180,E1 -6054.661,E2 -6054.661} C_VEL
LIN {X 0,Y 497.166,Z 596.406,A -85,B 0,C 180,E1 -6055.618,E2 -6055.618} C_VEL
LIN {X 0,Y 497.599,Z 585.066,A -85,B 0,C 180,E1 -6056.529,E2 -6056.529} C_VEL
LIN {X 0,Y 497.892,Z 574.212,A -85,B 0,C 180,E1 -6057.218,E2 -6057.218} C_VEL
LIN {X 0,Y 497.709,Z 569.413,A -85,B 0,C 180,E1 -6057.482,E2 -6057.482} C_VEL
LIN {X 0,Y 495.815,Z 562.727,A -85,B 0,C 180,E1 -6057.888,E2 -6057.888} C_VEL
LIN {X 0,Y 495.752,Z 562.733,A -85,B 0,C 180,E1 -6060.686,E2 -6060.686} C_VEL
LIN {X 0,Y 495.754,Z 562.733,A -85,B 0,C 180,E1 -6063.564,E2 -6063.564} C_VEL
LIN {X 0,Y 495.727,Z 562.737,A -85,B 0,C 180,E1 -6066.543,E2 -6066.543} C_VEL
LIN {X 0,Y 495.79,Z 562.73,A -85,B 0,C 180,E1 -6069.633,E2 -6069.633} C_VEL
LIN {X 0,Y 495.829,Z 562.863,A -85,B 0,C 180,E1 -6070.336,E2 -6070.336} C_VEL
LIN {X 0,Y 496.295,Z 567.72,A -85,B 0,C 180,E1 -6072.147,E2 -6072.147} C_VEL
LIN {X 0,Y 496.206,Z 575.709,A -85,B 0,C 180,E1 -6075.085,E2 -6075.085} C_VEL
LIN {X 0,Y 496.13,Z 583.145,A -85,B 0,C 180,E1 -6077.847,E2 -6077.847} C_VEL
LIN {X 0,Y 495.958,Z 591.247,A -85,B 0,C 180,E1 -6080.831,E2 -6080.831} C_VEL
LIN {X 0,Y 495.855,Z 599.458,A -85,B 0,C 180,E1 -6083.888,E2 -6083.888} C_VEL
LIN {X 0,Y 495.738,Z 607.175,A -85,B 0,C 180,E1 -6086.763,E2 -6086.763} C_VEL
LIN {X 0,Y 495.544,Z 615.585,A -85,B 0,C 180,E1 -6089.895,E2 -6089.895} C_VEL
LIN {X 0,Y 495.452,Z 622.744,A -85,B 0,C 180,E1 -6092.556,E2 -6092.556} C_VEL
LIN {X 0,Y 497.771,Z 636.049,A -85,B 0,C 180,E1 -6092.973,E2 -6092.973} C_VEL
LIN {X 0,Y 497.447,Z 648.919,A -85,B 0,C 180,E1 -6093.462,E2 -6093.462} C_VEL
LIN {X 0,Y 497.093,Z 661.32,A -85,B 0,C 180,E1 -6094.119,E2 -6094.119} C_VEL
LIN {X 0,Y 496.745,Z 672.523,A -85,B 0,C 180,E1 -6094.885,E2 -6094.885} C_VEL
LIN {X 0,Y 496.382,Z 682.742,A -85,B 0,C 180,E1 -6095.758,E2 -6095.758} C_VEL
LIN {X 0,Y 496.015,Z 692.293,A -85,B 0,C 180,E1 -6096.769,E2 -6096.769} C_VEL
LIN {X 0,Y 495.679,Z 701.233,A -85,B 0,C 180,E1 -6097.931,E2 -6097.931} C_VEL
LIN {X 0,Y 495.448,Z 708.014,A -85,B 0,C 180,E1 -6099.012,E2 -6099.012} C_VEL
LIN {X 0,Y 495.299,Z 713.57,A -85,B 0,C 180,E1 -6100.09,E2 -6100.09} C_VEL
LIN {X 0,Y 495.181,Z 718.915,A -85,B 0,C 180,E1 -6101.377,E2 -6101.377} C_VEL
LIN {X 0,Y 495.049,Z 722.96,A -85,B 0,C 180,E1 -6102.655,E2 -6102.655} C_VEL
LIN {X 0,Y 494.964,Z 725.014,A -85,B 0,C 180,E1 -6103.502,E2 -6103.502} C_VEL
LIN {X 0,Y 494.955,Z 727.436,A -85,B 0,C 180,E1 -6104.912,E2 -6104.912} C_VEL
LIN {X 0,Y 494.931,Z 728.489,A -85,B 0,C 180,E1 -6106.031,E2 -6106.031} C_VEL
LIN {X 0,Y 494.903,Z 728.797,A -85,B 0,C 180,E1 -6106.867,E2 -6106.867} C_VEL
LIN {X 0,Y 495.012,Z 728.268,A -85,B 0,C 180,E1 -6108.412,E2 -6108.412} C_VEL
LIN {X 0,Y 495.009,Z 727.214,A -85,B 0,C 180,E1 -6109.364,E2 -6109.364} C_VEL
LIN {X 0,Y 494.967,Z 725.887,A -85,B 0,C 180,E1 -6110.19,E2 -6110.19} C_VEL
LIN {X 0,Y 495.075,Z 723.048,A -85,B 0,C 180,E1 -6111.428,E2 -6111.428} C_VEL
LIN {X 0,Y 495.184,Z 719.187,A -85,B 0,C 180,E1 -6112.662,E2 -6112.662} C_VEL
LIN {X 0,Y 495.269,Z 714.201,A -85,B 0,C 180,E1 -6113.891,E2 -6113.891} C_VEL
LIN {X 0,Y 495.414,Z 707.913,A -85,B 0,C 180,E1 -6115.118,E2 -6115.118} C_VEL
LIN {X 0,Y 495.692,Z 700.1,A -85,B 0,C 180,E1 -6116.342,E2 -6116.342} C_VEL
LIN {X 0,Y 495.998,Z 692.146,A -85,B 0,C 180,E1 -6117.361,E2 -6117.361} C_VEL
LIN {X 0,Y 496.387,Z 682.447,A -85,B 0,C 180,E1 -6118.378,E2 -6118.378} C_VEL
LIN {X 0,Y 496.768,Z 671.571,A -85,B 0,C 180,E1 -6119.291,E2 -6119.291} C_VEL
LIN {X 0,Y 497.139,Z 661.025,A -85,B 0,C 180,E1 -6120,E2 -6120} C_VEL
LIN {X 0,Y 497.538,Z 648.349,A -85,B 0,C 180,E1 -6120.658,E2 -6120.658} C_VEL
LIN {X 0,Y 497.768,Z 635.539,A -85,B 0,C 180,E1 -6121.138,E2 -6121.138} C_VEL
LIN {X 0,Y 495.671,Z 624.299,A -85,B 0,C 180,E1 -6121.489,E2 -6121.489} C_VEL
LIN {X 0,Y 495.47,Z 623.28,A -85,B 0,C 180,E1 -6121.524,E2 -6121.524} C_VEL
LIN {X 0,Y 495.727,Z 614.225,A -85,B 0,C 180,E1 -6124.88,E2 -6124.88} C_VEL
LIN {X 0,Y 495.82,Z 605.338,A -85,B 0,C 180,E1 -6128.149,E2 -6128.149} C_VEL
LIN {X 0,Y 495.866,Z 599.673,A -85,B 0,C 180,E1 -6130.205,E2 -6130.205} C_VEL
LIN {X 0,Y 495.975,Z 592.723,A -85,B 0,C 180,E1 -6132.688,E2 -6132.688} C_VEL
LIN {X 0,Y 496,Z 584.101,A -85,B 0,C 180,E1 -6135.618,E2 -6135.618} C_VEL
LIN {X 0,Y 495.999,Z 575.063,A -85,B 0,C 180,E1 -6138.604,E2 -6138.604} C_VEL
LIN {X 0,Y 495.906,Z 565.486,A -85,B 0,C 180,E1 -6141.622,E2 -6141.622} C_VEL
LIN {X 0,Y 495.752,Z 562.736,A -85,B 0,C 180,E1 -6142.505,E2 -6142.505} C_VEL
LIN {X 0,Y 495.783,Z 562.734,A -85,B 0,C 180,E1 -6145.168,E2 -6145.168} C_VEL
LIN {X 0,Y 495.777,Z 562.733,A -85,B 0,C 180,E1 -6147.892,E2 -6147.892} C_VEL
LIN {X 0,Y 495.752,Z 562.735,A -85,B 0,C 180,E1 -6150.688,E2 -6150.688} C_VEL
LIN {X 0,Y 495.756,Z 562.734,A -85,B 0,C 180,E1 -6153.565,E2 -6153.565} C_VEL
LIN {X 0,Y 495.731,Z 562.737,A -85,B 0,C 180,E1 -6156.544,E2 -6156.544} C_VEL
LIN {X 0,Y 495.779,Z 562.731,A -85,B 0,C 180,E1 -6159.636,E2 -6159.636} C_VEL
LIN {X 0,Y 495.76,Z 562.733,A -85,B 0,C 180,E1 -6162.88,E2 -6162.88} C_VEL
LIN {X 0,Y 495.733,Z 562.736,A -85,B 0,C 180,E1 -6166,E2 -6166} C_VEL
LIN {X 0,Y 495.765,Z 562.733,A -85,B 0,C 180,E1 -6168.706,E2 -6168.706} C_VEL
LIN {X 0,Y 495.794,Z 562.771,A -85,B 0,C 180,E1 -6170.475,E2 -6170.475} C_VEL
LIN {X 0,Y 498.013,Z 574.095,A -85,B 0,C 180,E1 -6173.552,E2 -6173.552} C_VEL
LIN {X 0,Y 497.761,Z 584.455,A -85,B 0,C 180,E1 -6176.068,E2 -6176.068} C_VEL
LIN {X 0,Y 497.259,Z 598.914,A -85,B 0,C 180,E1 -6179.417,E2 -6179.417} C_VEL
LIN {X 0,Y 496.898,Z 613.374,A -85,B 0,C 180,E1 -6182.636,E2 -6182.636} C_VEL
LIN {X 0,Y 496.581,Z 625.939,A -85,B 0,C 180,E1 -6185.345,E2 -6185.345} C_VEL
LIN {X 0,Y 496.287,Z 639.386,A -85,B 0,C 180,E1 -6188.179,E2 -6188.179} C_VEL
LIN {X 0,Y 496.004,Z 654.929,A -85,B 0,C 180,E1 -6191.39,E2 -6191.39} C_VEL
LIN {X 0,Y 495.775,Z 668.532,A -85,B 0,C 180,E1 -6194.165,E2 -6194.165} C_VEL
LIN {X 0,Y 495.659,Z 674.829,A -85,B 0,C 180,E1 -6195.45,E2 -6195.45} C_VEL
LIN {X 0,Y 496.867,Z 685.366,A -85,B 0,C 180,E1 -6195.699,E2 -6195.699} C_VEL
LIN {X 0,Y 497.711,Z 692.611,A -85,B 0,C 180,E1 -6195.929,E2 -6195.929} C_VEL
LIN {X 0,Y 497.317,Z 705.27,A -85,B 0,C 180,E1 -6196.413,E2 -6196.413} C_VEL
LIN {X 0,Y 496.978,Z 717.007,A -85,B 0,C 180,E1 -6197.021,E2 -6197.021} C_VEL
LIN {X 0,Y 496.609,Z 727.951,A -85,B 0,C 180,E1 -6197.745,E2 -6197.745} C_VEL
LIN {X 0,Y 496.266,Z 739.05,A -85,B 0,C 180,E1 -6198.669,E2 -6198.669} C_VEL
LIN {X 0,Y 495.838,Z 749.925,A -85,B 0,C 180,E1 -6199.796,E2 -6199.796} C_VEL
LIN {X 0,Y 495.619,Z 757.982,A -85,B 0,C 180,E1 -6200.821,E2 -6200.821} C_VEL
LIN {X 0,Y 495.388,Z 765.868,A -85,B 0,C 180,E1 -6202.05,E2 -6202.05} C_VEL
LIN {X 0,Y 495.203,Z 773.145,A -85,B 0,C 180,E1 -6203.482,E2 -6203.482} C_VEL
LIN {X 0,Y 495.151,Z 778.001,A -85,B 0,C 180,E1 -6204.707,E2 -6204.707} C_VEL
LIN {X 0,Y 495.104,Z 781.709,A -85,B 0,C 180,E1 -6205.931,E2 -6205.931} C_VEL
LIN {X 0,Y 495.074,Z 783.622,A -85,B 0,C 180,E1 -6206.746,E2 -6206.746} C_VEL
LIN {X 0,Y 495.025,Z 785.064,A -85,B 0,C 180,E1 -6207.56,E2 -6207.56} C_VEL
LIN {X 0,Y 494.998,Z 786.087,A -85,B 0,C 180,E1 -6208.374,E2 -6208.374} C_VEL
LIN {X 0,Y 494.957,Z 786.706,A -85,B 0,C 180,E1 -6209.187,E2 -6209.187} C_VEL
LIN {X 0,Y 494.948,Z 786.924,A -85,B 0,C 180,E1 -6210.001,E2 -6210.001} C_VEL
LIN {X 0,Y 494.956,Z 786.711,A -85,B 0,C 180,E1 -6210.814,E2 -6210.814} C_VEL
LIN {X 0,Y 494.998,Z 786.088,A -85,B 0,C 180,E1 -6211.628,E2 -6211.628} C_VEL
LIN {X 0,Y 495.026,Z 785.06,A -85,B 0,C 180,E1 -6212.442,E2 -6212.442} C_VEL
LIN {X 0,Y 495.075,Z 783.619,A -85,B 0,C 180,E1 -6213.256,E2 -6213.256} C_VEL
LIN {X 0,Y 495.071,Z 780.606,A -85,B 0,C 180,E1 -6214.479,E2 -6214.479} C_VEL
LIN {X 0,Y 495.196,Z 776.545,A -85,B 0,C 180,E1 -6215.702,E2 -6215.702} C_VEL
LIN {X 0,Y 495.273,Z 770.385,A -85,B 0,C 180,E1 -6217.113,E2 -6217.113} C_VEL
LIN {X 0,Y 495.461,Z 763.432,A -85,B 0,C 180,E1 -6218.361,E2 -6218.361} C_VEL
LIN {X 0,Y 495.708,Z 754.99,A -85,B 0,C 180,E1 -6219.59,E2 -6219.59} C_VEL
LIN {X 0,Y 495.974,Z 746.331,A -85,B 0,C 180,E1 -6220.616,E2 -6220.616} C_VEL
LIN {X 0,Y 496.393,Z 735.675,A -85,B 0,C 180,E1 -6221.64,E2 -6221.64} C_VEL
LIN {X 0,Y 496.714,Z 724.569,A -85,B 0,C 180,E1 -6222.503,E2 -6222.503} C_VEL
LIN {X 0,Y 497.071,Z 713.635,A -85,B 0,C 180,E1 -6223.179,E2 -6223.179} C_VEL
LIN {X 0,Y 497.459,Z 701.849,A -85,B 0,C 180,E1 -6223.741,E2 -6223.741} C_VEL
LIN {X 0,Y 497.537,Z 690.115,A -85,B 0,C 180,E1 -6224.156,E2 -6224.156} C_VEL
LIN {X 0,Y 495.928,Z 678.439,A -85,B 0,C 180,E1 -6224.478,E2 -6224.478} C_VEL
LIN {X 0,Y 495.666,Z 674.947,A -85,B 0,C 180,E1 -6224.577,E2 -6224.577} C_VEL
LIN {X 0,Y 495.984,Z 658.53,A -85,B 0,C 180,E1 -6227.951,E2 -6227.951} C_VEL
LIN {X 0,Y 496.241,Z 642.999,A -85,B 0,C 180,E1 -6231.171,E2 -6231.171} C_VEL
LIN {X 0,Y 496.54,Z 628.548,A -85,B 0,C 180,E1 -6234.235,E2 -6234.235} C_VEL
LIN {X 0,Y 496.925,Z 614.066,A -85,B 0,C 180,E1 -6237.364,E2 -6237.364} C_VEL
LIN {X 0,Y 497.281,Z 600.18,A -85,B 0,C 180,E1 -6240.446,E2 -6240.446} C_VEL
LIN {X 0,Y 497.654,Z 588.171,A -85,B 0,C 180,E1 -6243.178,E2 -6243.178} C_VEL
LIN {X 0,Y 498.008,Z 575.725,A -85,B 0,C 180,E1 -6246.1,E2 -6246.1} C_VEL
LIN {X 0,Y 497.311,Z 570.435,A -85,B 0,C 180,E1 -6247.422,E2 -6247.422} C_VEL
LIN {X 0,Y 495.767,Z 562.733,A -85,B 0,C 180,E1 -6249.473,E2 -6249.473} C_VEL
LIN {X 0,Y 495.743,Z 562.735,A -85,B 0,C 180,E1 -6252.507,E2 -6252.507} C_VEL
LIN {X 0,Y 495.754,Z 562.734,A -85,B 0,C 180,E1 -6255.139,E2 -6255.139} C_VEL
LIN {X 0,Y 495.762,Z 562.733,A -85,B 0,C 180,E1 -6258.219,E2 -6258.219} C_VEL
LIN {X 0,Y 495.754,Z 562.733,A -85,B 0,C 180,E1 -6261.408,E2 -6261.408} C_VEL
LIN {X 0,Y 495.763,Z 562.732,A -85,B 0,C 180,E1 -6264.463,E2 -6264.463} C_VEL
LIN {X 0,Y 495.772,Z 562.731,A -85,B 0,C 180,E1 -6267.406,E2 -6267.406} C_VEL
LIN {X 0,Y 495.771,Z 562.731,A -85,B 0,C 180,E1 -6270.254,E2 -6270.254} C_VEL
LIN {X 0,Y 495.828,Z 562.724,A -85,B 0,C 180,E1 -6273.251,E2 -6273.251} C_VEL
LIN {X 0,Y 495.753,Z 562.734,A -85,B 0,C 180,E1 -6275.725,E2 -6275.725} C_VEL
LIN {X 0,Y 495.747,Z 562.734,A -85,B 0,C 180,E1 -6278.371,E2 -6278.371} C_VEL
LIN {X 0,Y 495.789,Z 562.729,A -85,B 0,C 180,E1 -6280.971,E2 -6280.971} C_VEL
LIN {X 0,Y 495.784,Z 562.729,A -85,B 0,C 180,E1 -6283.53,E2 -6283.53} C_VEL
LIN {X 0,Y 495.798,Z 562.73,A -85,B 0,C 180,E1 -6286.055,E2 -6286.055} C_VEL
LIN {X 0,Y 495.855,Z 562.721,A -85,B 0,C 180,E1 -6288.555,E2 -6288.555} C_VEL
LIN {X 0,Y 495.877,Z 562.719,A -85,B 0,C 180,E1 -6291.852,E2 -6291.852} C_VEL
LIN {X 0,Y 495.9,Z 562.717,A -85,B 0,C 180,E1 -6294.306,E2 -6294.306} C_VEL
LIN {X 0,Y 495.995,Z 562.703,A -85,B 0,C 180,E1 -6297.563,E2 -6297.563} C_VEL
LIN {X 0,Y 496.002,Z 562.703,A -85,B 0,C 180,E1 -6300,E2 -6300} C_VEL
LIN {X 0,Y 495.996,Z 562.705,A -85,B 0,C 180,E1 -6302.436,E2 -6302.436} C_VEL
LIN {X 0,Y 495.899,Z 562.714,A -85,B 0,C 180,E1 -6305.693,E2 -6305.693} C_VEL
LIN {X 0,Y 495.876,Z 562.719,A -85,B 0,C 180,E1 -6308.148,E2 -6308.148} C_VEL
LIN {X 0,Y 495.854,Z 562.72,A -85,B 0,C 180,E1 -6311.445,E2 -6311.445} C_VEL
LIN {X 0,Y 495.793,Z 562.729,A -85,B 0,C 180,E1 -6314.782,E2 -6314.782} C_VEL
LIN {X 0,Y 495.79,Z 562.729,A -85,B 0,C 180,E1 -6317.318,E2 -6317.318} C_VEL
LIN {X 0,Y 495.774,Z 562.731,A -85,B 0,C 180,E1 -6319.89,E2 -6319.89} C_VEL
LIN {X 0,Y 495.768,Z 562.732,A -85,B 0,C 180,E1 -6322.862,E2 -6322.862} C_VEL
LIN {X 0,Y 495.793,Z 562.729,A -85,B 0,C 180,E1 -6326.067,E2 -6326.067} C_VEL
LIN {X 0,Y 495.774,Z 562.731,A -85,B 0,C 180,E1 -6328.814,E2 -6328.814} C_VEL
LIN {X 0,Y 495.758,Z 562.733,A -85,B 0,C 180,E1 -6331.725,E2 -6331.725} C_VEL
LIN {X 0,Y 495.778,Z 562.731,A -85,B 0,C 180,E1 -6334.695,E2 -6334.695} C_VEL
LIN {X 0,Y 495.733,Z 562.736,A -85,B 0,C 180,E1 -6337.561,E2 -6337.561} C_VEL
LIN {X 0,Y 495.768,Z 562.733,A -85,B 0,C 180,E1 -6340.699,E2 -6340.699} C_VEL
LIN {X 0,Y 495.736,Z 562.735,A -85,B 0,C 180,E1 -6343.695,E2 -6343.695} C_VEL
LIN {X 0,Y 495.736,Z 562.736,A -85,B 0,C 180,E1 -6346.304,E2 -6346.304} C_VEL
LIN {X 0,Y 495.768,Z 562.73,A -85,B 0,C 180,E1 -6349.3,E2 -6349.3} C_VEL
LIN {X 0,Y 495.73,Z 562.738,A -85,B 0,C 180,E1 -6352.438,E2 -6352.438} C_VEL
LIN {X 0,Y 495.778,Z 562.728,A -85,B 0,C 180,E1 -6355.456,E2 -6355.456} C_VEL
LIN {X 0,Y 495.76,Z 562.734,A -85,B 0,C 180,E1 -6358.363,E2 -6358.363} C_VEL
LIN {X 0,Y 495.754,Z 562.731,A -85,B 0,C 180,E1 -6360.757,E2 -6360.757} C_VEL
LIN {X 0,Y 495.096,Z 562.814,A -85,B 0,C 180,E1 -6361.436,E2 -6361.436} C_VEL
LIN {X 0,Y 492.24,Z 563.171,A -85,B 0,C 180,E1 -6362.539,E2 -6362.539} C_VEL
LIN {X 0,Y 489.831,Z 563.469,A -85,B 0,C 180,E1 -6363.427,E2 -6363.427} C_VEL
LIN {X 0,Y 488.815,Z 563.598,A -85,B 0,C 180,E1 -6364.114,E2 -6364.114} C_VEL
LIN {X 0,Y 488.743,Z 563.607,A -85,B 0,C 180,E1 -6364.346,E2 -6364.346} C_VEL
LIN {X 0,Y 488.721,Z 563.608,A -85,B 0,C 180,E1 -6367.152,E2 -6367.152} C_VEL
LIN {X 0,Y 488.725,Z 563.607,A -85,B 0,C 180,E1 -6369.81,E2 -6369.81} C_VEL
LIN {X 0,Y 488.735,Z 563.61,A -85,B 0,C 180,E1 -6372.423,E2 -6372.423} C_VEL
LIN {X 0,Y 488.762,Z 563.604,A -85,B 0,C 180,E1 -6374.999,E2 -6374.999} C_VEL
LIN {X 0,Y 488.83,Z 563.598,A -85,B 0,C 180,E1 -6378.387,E2 -6378.387} C_VEL
LIN {X 0,Y 488.817,Z 563.597,A -85,B 0,C 180,E1 -6381.733,E2 -6381.733} C_VEL
LIN {X 0,Y 488.855,Z 563.594,A -85,B 0,C 180,E1 -6384.224,E2 -6384.224} C_VEL
LIN {X 0,Y 488.962,Z 563.581,A -85,B 0,C 180,E1 -6387.528,E2 -6387.528} C_VEL
LIN {X 0,Y 488.968,Z 563.581,A -85,B 0,C 180,E1 -6390.051,E2 -6390.051} C_VEL
LIN {X 0,Y 490.95,Z 571.497,A -85,B 0,C 180,E1 -6390.512,E2 -6390.512} C_VEL
LIN {X 0,Y 490.73,Z 583.412,A -85,B 0,C 180,E1 -6391.23,E2 -6391.23} C_VEL
LIN {X 0,Y 490.404,Z 594.132,A -85,B 0,C 180,E1 -6392.052,E2 -6392.052} C_VEL
LIN {X 0,Y 490.054,Z 602.877,A -85,B 0,C 180,E1 -6392.876,E2 -6392.876} C_VEL
LIN {X 0,Y 489.725,Z 611.848,A -85,B 0,C 180,E1 -6393.908,E2 -6393.908} C_VEL
LIN {X 0,Y 489.319,Z 620.615,A -85,B 0,C 180,E1 -6395.149,E2 -6395.149} C_VEL
LIN {X 0,Y 489.13,Z 627.645,A -85,B 0,C 180,E1 -6396.393,E2 -6396.393} C_VEL
LIN {X 0,Y 488.889,Z 632.428,A -85,B 0,C 180,E1 -6397.433,E2 -6397.433} C_VEL
LIN {X 0,Y 488.697,Z 637.073,A -85,B 0,C 180,E1 -6398.684,E2 -6398.684} C_VEL
LIN {X 0,Y 488.53,Z 640.633,A -85,B 0,C 180,E1 -6399.94,E2 -6399.94} C_VEL
LIN {X 0,Y 488.449,Z 642.463,A -85,B 0,C 180,E1 -6400.78,E2 -6400.78} C_VEL
LIN {X 0,Y 488.425,Z 644.214,A -85,B 0,C 180,E1 -6401.916,E2 -6401.916} C_VEL
LIN {X 0,Y 488.359,Z 645.381,A -85,B 0,C 180,E1 -6403.311,E2 -6403.311} C_VEL
LIN {X 0,Y 488.361,Z 645.535,A -85,B 0,C 180,E1 -6404.16,E2 -6404.16} C_VEL
LIN {X 0,Y 488.39,Z 645.055,A -85,B 0,C 180,E1 -6405.392,E2 -6405.392} C_VEL
LIN {X 0,Y 488.429,Z 643.552,A -85,B 0,C 180,E1 -6406.724,E2 -6406.724} C_VEL
LIN {X 0,Y 488.58,Z 640.361,A -85,B 0,C 180,E1 -6408.309,E2 -6408.309} C_VEL
LIN {X 0,Y 488.74,Z 636.108,A -85,B 0,C 180,E1 -6409.75,E2 -6409.75} C_VEL
LIN {X 0,Y 488.981,Z 630.95,A -85,B 0,C 180,E1 -6411.057,E2 -6411.057} C_VEL
LIN {X 0,Y 489.262,Z 624.293,A -85,B 0,C 180,E1 -6412.373,E2 -6412.373} C_VEL
LIN {X 0,Y 489.66,Z 615.863,A -85,B 0,C 180,E1 -6413.695,E2 -6413.695} C_VEL
LIN {X 0,Y 489.984,Z 607.168,A -85,B 0,C 180,E1 -6414.793,E2 -6414.793} C_VEL
LIN {X 0,Y 490.315,Z 597.184,A -85,B 0,C 180,E1 -6415.809,E2 -6415.809} C_VEL
LIN {X 0,Y 490.739,Z 586.238,A -85,B 0,C 180,E1 -6416.7,E2 -6416.7} C_VEL
LIN {X 0,Y 491.051,Z 574.378,A -85,B 0,C 180,E1 -6417.458,E2 -6417.458} C_VEL
LIN {X 0,Y 490.983,Z 571.31,A -85,B 0,C 180,E1 -6417.627,E2 -6417.627} C_VEL
LIN {X 0,Y 488.771,Z 563.605,A -85,B 0,C 180,E1 -6418.087,E2 -6418.087} C_VEL
LIN {X 0,Y 488.691,Z 563.61,A -85,B 0,C 180,E1 -6421.179,E2 -6421.179} C_VEL
LIN {X 0,Y 488.727,Z 563.608,A -85,B 0,C 180,E1 -6424.112,E2 -6424.112} C_VEL
LIN {X 0,Y 488.677,Z 563.615,A -85,B 0,C 180,E1 -6427.158,E2 -6427.158} C_VEL
LIN {X 0,Y 488.781,Z 563.719,A -85,B 0,C 180,E1 -6430.182,E2 -6430.182} C_VEL
LIN {X 0,Y 489.298,Z 568.576,A -85,B 0,C 180,E1 -6432.023,E2 -6432.023} C_VEL
LIN {X 0,Y 489.218,Z 575.89,A -85,B 0,C 180,E1 -6434.741,E2 -6434.741} C_VEL
LIN {X 0,Y 489.138,Z 583.411,A -85,B 0,C 180,E1 -6437.523,E2 -6437.523} C_VEL
LIN {X 0,Y 488.986,Z 590.695,A -85,B 0,C 180,E1 -6440.24,E2 -6440.24} C_VEL
LIN {X 0,Y 488.868,Z 598.839,A -85,B 0,C 180,E1 -6443.279,E2 -6443.279} C_VEL
LIN {X 0,Y 488.727,Z 607.468,A -85,B 0,C 180,E1 -6446.515,E2 -6446.515} C_VEL
LIN {X 0,Y 488.521,Z 616.14,A -85,B 0,C 180,E1 -6449.767,E2 -6449.767} C_VEL
LIN {X 0,Y 488.439,Z 623.254,A -85,B 0,C 180,E1 -6452.36,E2 -6452.36} C_VEL
LIN {X 0,Y 490.795,Z 635.958,A -85,B 0,C 180,E1 -6452.761,E2 -6452.761} C_VEL
LIN {X 0,Y 490.577,Z 648.601,A -85,B 0,C 180,E1 -6453.246,E2 -6453.246} C_VEL
LIN {X 0,Y 490.256,Z 660.083,A -85,B 0,C 180,E1 -6453.845,E2 -6453.845} C_VEL
LIN {X 0,Y 489.829,Z 672.286,A -85,B 0,C 180,E1 -6454.675,E2 -6454.675} C_VEL
LIN {X 0,Y 489.407,Z 683.211,A -85,B 0,C 180,E1 -6455.616,E2 -6455.616} C_VEL
LIN {X 0,Y 489.021,Z 692.771,A -85,B 0,C 180,E1 -6456.644,E2 -6456.644} C_VEL
LIN {X 0,Y 488.673,Z 701.684,A -85,B 0,C 180,E1 -6457.82,E2 -6457.82} C_VEL
LIN {X 0,Y 488.433,Z 708.46,A -85,B 0,C 180,E1 -6458.917,E2 -6458.917} C_VEL
LIN {X 0,Y 488.231,Z 714.995,A -85,B 0,C 180,E1 -6460.228,E2 -6460.228} C_VEL
LIN {X 0,Y 488.111,Z 720.084,A -85,B 0,C 180,E1 -6461.533,E2 -6461.533} C_VEL
LIN {X 0,Y 487.966,Z 723.934,A -85,B 0,C 180,E1 -6462.828,E2 -6462.828} C_VEL
LIN {X 0,Y 487.862,Z 726.678,A -85,B 0,C 180,E1 -6464.115,E2 -6464.115} C_VEL
LIN {X 0,Y 487.881,Z 727.95,A -85,B 0,C 180,E1 -6464.972,E2 -6464.972} C_VEL
LIN {X 0,Y 487.854,Z 728.778,A -85,B 0,C 180,E1 -6465.824,E2 -6465.824} C_VEL
LIN {X 0,Y 487.827,Z 729.163,A -85,B 0,C 180,E1 -6466.673,E2 -6466.673} C_VEL
LIN {X 0,Y 487.843,Z 729.153,A -85,B 0,C 180,E1 -6467.521,E2 -6467.521} C_VEL
LIN {X 0,Y 487.936,Z 728.735,A -85,B 0,C 180,E1 -6468.367,E2 -6468.367} C_VEL
LIN {X 0,Y 487.918,Z 727.873,A -85,B 0,C 180,E1 -6469.208,E2 -6469.208} C_VEL
LIN {X 0,Y 487.898,Z 726.618,A -85,B 0,C 180,E1 -6470.046,E2 -6470.046} C_VEL
LIN {X 0,Y 487.982,Z 723.927,A -85,B 0,C 180,E1 -6471.303,E2 -6471.303} C_VEL
LIN {X 0,Y 488.112,Z 720.216,A -85,B 0,C 180,E1 -6472.555,E2 -6472.555} C_VEL
LIN {X 0,Y 488.219,Z 714.853,A -85,B 0,C 180,E1 -6473.931,E2 -6473.931} C_VEL
LIN {X 0,Y 488.391,Z 708.175,A -85,B 0,C 180,E1 -6475.254,E2 -6475.254} C_VEL
LIN {X 0,Y 488.691,Z 700.325,A -85,B 0,C 180,E1 -6476.496,E2 -6476.496} C_VEL
LIN {X 0,Y 489.033,Z 692.323,A -85,B 0,C 180,E1 -6477.529,E2 -6477.529} C_VEL
LIN {X 0,Y 489.444,Z 682.543,A -85,B 0,C 180,E1 -6478.56,E2 -6478.56} C_VEL
LIN {X 0,Y 489.851,Z 671.602,A -85,B 0,C 180,E1 -6479.487,E2 -6479.487} C_VEL
LIN {X 0,Y 490.23,Z 660.977,A -85,B 0,C 180,E1 -6480.206,E2 -6480.206} C_VEL
LIN {X 0,Y 490.638,Z 649.282,A -85,B 0,C 180,E1 -6480.821,E2 -6480.821} C_VEL
LIN {X 0,Y 490.824,Z 635.95,A -85,B 0,C 180,E1 -6481.334,E2 -6481.334} C_VEL
LIN {X 0,Y 488.807,Z 625.43,A -85,B 0,C 180,E1 -6481.674,E2 -6481.674} C_VEL
LIN {X 0,Y 488.461,Z 623.649,A -85,B 0,C 180,E1 -6481.752,E2 -6481.752} C_VEL
LIN {X 0,Y 488.702,Z 615.045,A -85,B 0,C 180,E1 -6484.95,E2 -6484.95} C_VEL
LIN {X 0,Y 488.801,Z 606.07,A -85,B 0,C 180,E1 -6488.267,E2 -6488.267} C_VEL
LIN {X 0,Y 488.946,Z 598.113,A -85,B 0,C 180,E1 -6491.189,E2 -6491.189} C_VEL
LIN {X 0,Y 488.968,Z 589.625,A -85,B 0,C 180,E1 -6494.143,E2 -6494.143} C_VEL
LIN {X 0,Y 489.01,Z 580.731,A -85,B 0,C 180,E1 -6497.135,E2 -6497.135} C_VEL
LIN {X 0,Y 488.933,Z 571.381,A -85,B 0,C 180,E1 -6500.181,E2 -6500.181} C_VEL
LIN {X 0,Y 488.823,Z 564.244,A -85,B 0,C 180,E1 -6502.396,E2 -6502.396} C_VEL
LIN {X 0,Y 488.717,Z 563.612,A -85,B 0,C 180,E1 -6502.624,E2 -6502.624} C_VEL
LIN {X 0,Y 488.745,Z 563.61,A -85,B 0,C 180,E1 -6505.556,E2 -6505.556} C_VEL
LIN {X 0,Y 488.741,Z 563.609,A -85,B 0,C 180,E1 -6508.329,E2 -6508.329} C_VEL
LIN {X 0,Y 488.691,Z 563.615,A -85,B 0,C 180,E1 -6511.18,E2 -6511.18} C_VEL
LIN {X 0,Y 488.73,Z 563.609,A -85,B 0,C 180,E1 -6514.113,E2 -6514.113} C_VEL
LIN {X 0,Y 488.68,Z 563.614,A -85,B 0,C 180,E1 -6517.159,E2 -6517.159} C_VEL
LIN {X 0,Y 488.738,Z 563.608,A -85,B 0,C 180,E1 -6519.251,E2 -6519.251} C_VEL
LIN {X 0,Y 488.731,Z 563.606,A -85,B 0,C 180,E1 -6522.522,E2 -6522.522} C_VEL
LIN {X 0,Y 488.699,Z 563.613,A -85,B 0,C 180,E1 -6525.977,E2 -6525.977} C_VEL
LIN {X 0,Y 488.72,Z 563.609,A -85,B 0,C 180,E1 -6528.587,E2 -6528.587} C_VEL
LIN {X 0,Y 488.763,Z 563.716,A -85,B 0,C 180,E1 -6530.186,E2 -6530.186} C_VEL
LIN {X 0,Y 490.967,Z 574.862,A -85,B 0,C 180,E1 -6533.285,E2 -6533.285} C_VEL
LIN {X 0,Y 491.03,Z 580.355,A -85,B 0,C 180,E1 -6534.67,E2 -6534.67} C_VEL
LIN {X 0,Y 490.563,Z 591.7,A -85,B 0,C 180,E1 -6537.414,E2 -6537.414} C_VEL
LIN {X 0,Y 490.117,Z 605.364,A -85,B 0,C 180,E1 -6540.587,E2 -6540.587} C_VEL
LIN {X 0,Y 489.741,Z 618.782,A -85,B 0,C 180,E1 -6543.586,E2 -6543.586} C_VEL
LIN {X 0,Y 489.381,Z 633.545,A -85,B 0,C 180,E1 -6546.796,E2 -6546.796} C_VEL
LIN {X 0,Y 489.043,Z 648.841,A -85,B 0,C 180,E1 -6550.044,E2 -6550.044} C_VEL
LIN {X 0,Y 488.756,Z 663.357,A -85,B 0,C 180,E1 -6553.072,E2 -6553.072} C_VEL
LIN {X 0,Y 488.597,Z 673.769,A -85,B 0,C 180,E1 -6555.235,E2 -6555.235} C_VEL
LIN {X 0,Y 489.834,Z 685.743,A -85,B 0,C 180,E1 -6555.529,E2 -6555.529} C_VEL
LIN {X 0,Y 490.756,Z 693.085,A -85,B 0,C 180,E1 -6555.778,E2 -6555.778} C_VEL
LIN {X 0,Y 490.343,Z 705.349,A -85,B 0,C 180,E1 -6556.269,E2 -6556.269} C_VEL
LIN {X 0,Y 489.992,Z 716.239,A -85,B 0,C 180,E1 -6556.85,E2 -6556.85} C_VEL
LIN {X 0,Y 489.566,Z 728.234,A -85,B 0,C 180,E1 -6557.671,E2 -6557.671} C_VEL
LIN {X 0,Y 489.186,Z 739.082,A -85,B 0,C 180,E1 -6558.608,E2 -6558.608} C_VEL
LIN {X 0,Y 488.797,Z 748.874,A -85,B 0,C 180,E1 -6559.647,E2 -6559.647} C_VEL
LIN {X 0,Y 488.552,Z 756.932,A -85,B 0,C 180,E1 -6560.687,E2 -6560.687} C_VEL
LIN {X 0,Y 488.339,Z 764.831,A -85,B 0,C 180,E1 -6561.935,E2 -6561.935} C_VEL
LIN {X 0,Y 488.141,Z 772.107,A -85,B 0,C 180,E1 -6563.387,E2 -6563.387} C_VEL
LIN {X 0,Y 488.094,Z 776.977,A -85,B 0,C 180,E1 -6564.63,E2 -6564.63} C_VEL
LIN {X 0,Y 488.042,Z 780.685,A -85,B 0,C 180,E1 -6565.872,E2 -6565.872} C_VEL
LIN {X 0,Y 488.029,Z 782.598,A -85,B 0,C 180,E1 -6566.699,E2 -6566.699} C_VEL
LIN {X 0,Y 487.987,Z 784.055,A -85,B 0,C 180,E1 -6567.524,E2 -6567.524} C_VEL
LIN {X 0,Y 487.964,Z 785.081,A -85,B 0,C 180,E1 -6568.35,E2 -6568.35} C_VEL
LIN {X 0,Y 487.927,Z 785.7,A -85,B 0,C 180,E1 -6569.175,E2 -6569.175} C_VEL
LIN {X 0,Y 487.92,Z 785.914,A -85,B 0,C 180,E1 -6570.001,E2 -6570.001} C_VEL
LIN {X 0,Y 487.926,Z 785.707,A -85,B 0,C 180,E1 -6570.826,E2 -6570.826} C_VEL
LIN {X 0,Y 487.964,Z 785.082,A -85,B 0,C 180,E1 -6571.651,E2 -6571.651} C_VEL
LIN {X 0,Y 487.99,Z 784.039,A -85,B 0,C 180,E1 -6572.477,E2 -6572.477} C_VEL
LIN {X 0,Y 488.03,Z 782.594,A -85,B 0,C 180,E1 -6573.303,E2 -6573.303} C_VEL
LIN {X 0,Y 488.021,Z 779.589,A -85,B 0,C 180,E1 -6574.544,E2 -6574.544} C_VEL
LIN {X 0,Y 488.139,Z 775.526,A -85,B 0,C 180,E1 -6575.785,E2 -6575.785} C_VEL
LIN {X 0,Y 488.191,Z 769.272,A -85,B 0,C 180,E1 -6577.237,E2 -6577.237} C_VEL
LIN {X 0,Y 488.425,Z 762.417,A -85,B 0,C 180,E1 -6578.482,E2 -6578.482} C_VEL
LIN {X 0,Y 488.648,Z 753.973,A -85,B 0,C 180,E1 -6579.73,E2 -6579.73} C_VEL
LIN {X 0,Y 488.936,Z 745.315,A -85,B 0,C 180,E1 -6580.77,E2 -6580.77} C_VEL
LIN {X 0,Y 489.389,Z 734.661,A -85,B 0,C 180,E1 -6581.809,E2 -6581.809} C_VEL
LIN {X 0,Y 489.73,Z 723.412,A -85,B 0,C 180,E1 -6582.694,E2 -6582.694} C_VEL
LIN {X 0,Y 490.106,Z 712.621,A -85,B 0,C 180,E1 -6583.37,E2 -6583.37} C_VEL
LIN {X 0,Y 490.512,Z 700.833,A -85,B 0,C 180,E1 -6583.94,E2 -6583.94} C_VEL
LIN {X 0,Y 490.581,Z 690.878,A -85,B 0,C 180,E1 -6584.308,E2 -6584.308} C_VEL
LIN {X 0,Y 489.032,Z 678.922,A -85,B 0,C 180,E1 -6584.66,E2 -6584.66} C_VEL
LIN {X 0,Y 488.583,Z 673.919,A -85,B 0,C 180,E1 -6584.793,E2 -6584.793} C_VEL
LIN {X 0,Y 488.914,Z 657.571,A -85,B 0,C 180,E1 -6588.209,E2 -6588.209} C_VEL
LIN {X 0,Y 489.173,Z 643.144,A -85,B 0,C 180,E1 -6591.271,E2 -6591.271} C_VEL
LIN {X 0,Y 489.504,Z 628.716,A -85,B 0,C 180,E1 -6594.38,E2 -6594.38} C_VEL
LIN {X 0,Y 489.881,Z 615.33,A -85,B 0,C 180,E1 -6597.329,E2 -6597.329} C_VEL
LIN {X 0,Y 490.268,Z 601.655,A -85,B 0,C 180,E1 -6600.4,E2 -6600.4} C_VEL
LIN {X 0,Y 490.692,Z 588.628,A -85,B 0,C 180,E1 -6603.407,E2 -6603.407} C_VEL
LIN {X 0,Y 491.049,Z 576.448,A -85,B 0,C 180,E1 -6606.311,E2 -6606.311} C_VEL
LIN {X 0,Y 489.905,Z 569.56,A -85,B 0,C 180,E1 -6608.088,E2 -6608.088} C_VEL
LIN {X 0,Y 488.718,Z 563.612,A -85,B 0,C 180,E1 -6609.72,E2 -6609.72} C_VEL
LIN {X 0,Y 488.715,Z 563.611,A -85,B 0,C 180,E1 -6612.827,E2 -6612.827} C_VEL
LIN {X 0,Y 488.705,Z 563.612,A -85,B 0,C 180,E1 -6615.976,E2 -6615.976} C_VEL
LIN {X 0,Y 488.713,Z 563.611,A -85,B 0,C 180,E1 -6618.585,E2 -6618.585} C_VEL
LIN {X 0,Y 488.708,Z 563.61,A -85,B 0,C 180,E1 -6620.947,E2 -6620.947} C_VEL
LIN {X 0,Y 488.69,Z 563.614,A -85,B 0,C 180,E1 -6623.869,E2 -6623.869} C_VEL
LIN {X 0,Y 488.743,Z 563.607,A -85,B 0,C 180,E1 -6626.877,E2 -6626.877} C_VEL
LIN {X 0,Y 488.728,Z 563.609,A -85,B 0,C 180,E1 -6629.781,E2 -6629.781} C_VEL
LIN {X 0,Y 488.797,Z 563.6,A -85,B 0,C 180,E1 -6633.056,E2 -6633.056} C_VEL
LIN {X 0,Y 488.693,Z 563.613,A -85,B 0,C 180,E1 -6636.254,E2 -6636.254} C_VEL
LIN {X 0,Y 488.751,Z 563.605,A -85,B 0,C 180,E1 -6639.176,E2 -6639.176} C_VEL
LIN {X 0,Y 488.739,Z 563.609,A -85,B 0,C 180,E1 -6642.423,E2 -6642.423} C_VEL
LIN {X 0,Y 488.766,Z 563.603,A -85,B 0,C 180,E1 -6644.999,E2 -6644.999} C_VEL
LIN {X 0,Y 488.809,Z 563.6,A -85,B 0,C 180,E1 -6648.387,E2 -6648.387} C_VEL
LIN {X 0,Y 488.822,Z 563.596,A -85,B 0,C 180,E1 -6651.733,E2 -6651.733} C_VEL
LIN {X 0,Y 488.859,Z 563.594,A -85,B 0,C 180,E1 -6654.224,E2 -6654.224} C_VEL
LIN {X 0,Y 488.963,Z 563.578,A -85,B 0,C 180,E1 -6657.528,E2 -6657.528} C_VEL
LIN {X 0,Y 488.958,Z 563.581,A -85,B 0,C 180,E1 -6660.823,E2 -6660.823} C_VEL
LIN {X 0,Y 488.963,Z 563.581,A -85,B 0,C 180,E1 -6662.471,E2 -6662.471} C_VEL
LIN {X 0,Y 488.859,Z 563.592,A -85,B 0,C 180,E1 -6665.775,E2 -6665.775} C_VEL
LIN {X 0,Y 488.82,Z 563.599,A -85,B 0,C 180,E1 -6668.266,E2 -6668.266} C_VEL
LIN {X 0,Y 488.808,Z 563.598,A -85,B 0,C 180,E1 -6671.612,E2 -6671.612} C_VEL
LIN {X 0,Y 488.765,Z 563.605,A -85,B 0,C 180,E1 -6675,E2 -6675} C_VEL
LIN {X 0,Y 488.758,Z 563.606,A -85,B 0,C 180,E1 -6678.442,E2 -6678.442} C_VEL
LIN {X 0,Y 488.71,Z 563.61,A -85,B 0,C 180,E1 -6681.07,E2 -6681.07} C_VEL
LIN {X 0,Y 488.696,Z 563.612,A -85,B 0,C 180,E1 -6683.745,E2 -6683.745} C_VEL
LIN {X 0,Y 488.794,Z 563.6,A -85,B 0,C 180,E1 -6686.943,E2 -6686.943} C_VEL
LIN {X 0,Y 488.712,Z 563.613,A -85,B 0,C 180,E1 -6690.362,E2 -6690.362} C_VEL
LIN {X 0,Y 488.738,Z 563.606,A -85,B 0,C 180,E1 -6693.484,E2 -6693.484} C_VEL
LIN {X 0,Y 488.691,Z 563.615,A -85,B 0,C 180,E1 -6696.355,E2 -6696.355} C_VEL
LIN {X 0,Y 488.703,Z 563.611,A -85,B 0,C 180,E1 -6699.254,E2 -6699.254} C_VEL
LIN {X 0,Y 488.725,Z 563.607,A -85,B 0,C 180,E1 -6701.601,E2 -6701.601} C_VEL
LIN {X 0,Y 488.713,Z 563.61,A -85,B 0,C 180,E1 -6704.801,E2 -6704.801} C_VEL
LIN {X 0,Y 488.696,Z 563.611,A -85,B 0,C 180,E1 -6707.474,E2 -6707.474} C_VEL
LIN {X 0,Y 488.734,Z 563.606,A -85,B 0,C 180,E1 -6709.676,E2 -6709.676} C_VEL
LIN {X 0,Y 488.68,Z 563.614,A -85,B 0,C 180,E1 -6712.841,E2 -6712.841} C_VEL
LIN {X 0,Y 488.731,Z 563.607,A -85,B 0,C 180,E1 -6715.887,E2 -6715.887} C_VEL
LIN {X 0,Y 488.695,Z 563.613,A -85,B 0,C 180,E1 -6718.82,E2 -6718.82} C_VEL
LIN {X 0,Y 488.745,Z 563.605,A -85,B 0,C 180,E1 -6721.671,E2 -6721.671} C_VEL
LIN {X 0,Y 488.743,Z 563.607,A -85,B 0,C 180,E1 -6724.346,E2 -6724.346} C_VEL
LIN {X 0,Y 488.099,Z 563.692,A -85,B 0,C 180,E1 -6725.034,E2 -6725.034} C_VEL
LIN {X 0,Y 485.23,Z 564.05,A -85,B 0,C 180,E1 -6726.15,E2 -6726.15} C_VEL
LIN {X 0,Y 482.784,Z 564.35,A -85,B 0,C 180,E1 -6727.05,E2 -6727.05} C_VEL
LIN {X 0,Y 481.726,Z 564.48,A -85,B 0,C 180,E1 -6727.745,E2 -6727.745} C_VEL
LIN {X 0,Y 481.637,Z 564.49,A -85,B 0,C 180,E1 -6727.981,E2 -6727.981} C_VEL
LIN {X 0,Y 481.706,Z 564.484,A -85,B 0,C 180,E1 -6730.392,E2 -6730.392} C_VEL
LIN {X 0,Y 481.691,Z 564.485,A -85,B 0,C 180,E1 -6733.033,E2 -6733.033} C_VEL
LIN {X 0,Y 481.69,Z 564.484,A -85,B 0,C 180,E1 -6735.638,E2 -6735.638} C_VEL
LIN {X 0,Y 481.795,Z 564.473,A -85,B 0,C 180,E1 -6738.215,E2 -6738.215} C_VEL
LIN {X 0,Y 481.762,Z 564.475,A -85,B 0,C 180,E1 -6741.611,E2 -6741.611} C_VEL
LIN {X 0,Y 481.816,Z 564.47,A -85,B 0,C 180,E1 -6744.139,E2 -6744.139} C_VEL
LIN {X 0,Y 481.928,Z 564.457,A -85,B 0,C 180,E1 -6747.492,E2 -6747.492} C_VEL
LIN {X 0,Y 481.942,Z 564.656,A -85,B 0,C 180,E1 -6749.869,E2 -6749.869} C_VEL
LIN {X 0,Y 484.007,Z 572.259,A -85,B 0,C 180,E1 -6750.311,E2 -6750.311} C_VEL
LIN {X 0,Y 483.957,Z 581.096,A -85,B 0,C 180,E1 -6750.831,E2 -6750.831} C_VEL
LIN {X 0,Y 483.6,Z 592.453,A -85,B 0,C 180,E1 -6751.665,E2 -6751.665} C_VEL
